SYSTEM VerticalCoalMill
  (* Version 1.0, Author, 4DIAC-Consortium *)
  APPLICATION Process
    FBS
      mF : REAL2REAL(IN := 1);
      F_MUL : F_MUL;
      F_ADD : F_ADD;
      F_ADD_0 : F_ADD;
      F_SUB : F_SUB;
      REAL2REAL_0 : REAL2REAL;
      REAL2REAL_0_0 : REAL2REAL;
      REAL2REAL_0_1 : REAL2REAL;
      a1 : REAL2REAL(IN := 0.5);
      m_SB : REAL2REAL(IN := 1);
      m_CB : REAL2REAL(IN := 1);
      E_CYCLE : E_CYCLE(DT := T#200ms);
      FB_INTEGRATE : FB_INTEGRATE(K := 1);
      REAL2REAL_0_1_0 : REAL2REAL;
      M_B2 : REAL2REAL;
      F_DIV : F_DIV;
      mBG : REAL2REAL;
      tauBG : REAL2REAL(IN := 0.5);
      MV_from_ESCADA : SUBSCRIBE_1(QI := 1, ID := 127.0.0.1:63100);
      PP_from_ESCADA1 : SUBSCRIBE_2(QI := 1, ID := 127.0.0.1:64100);
      START_Subscribe : SUBSCRIBE_1(QI := 1, ID := 127.0.0.1:10000);
      E_SWITCH_0 : E_SWITCH;
      m_BG : REAL2REAL(IN := 1);
      gamma1 : REAL2REAL(IN := 0.5);
      bJ : REAL2REAL(IN := 0.5);
      gammaJ : REAL2REAL(IN := 0.5);
      F_ADD_1 : F_ADD;
      REAL2REAL_2_0 : REAL2REAL;
      F_SUB_0 : F_SUB;
      FB_INTEGRATE_0 : FB_INTEGRATE(K := 1);
      REAL2REAL_2_0_0 : REAL2REAL;
      F_DIV_0 : F_DIV;
      tauGS : REAL2REAL(IN := 0.5);
      mGS : REAL2REAL;
      E_CYCLE_0 : E_CYCLE(DT := T#200ms);
      F_MUL_1 : F_MUL;
      F_MUL_1_2 : F_MUL;
      F_MUL_1_3 : F_MUL;
      REAL2REAL_2_0_3 : REAL2REAL;
      F_SUB_0_0 : F_SUB;
      REAL2REAL_2_0_3_0 : REAL2REAL;
      REAL2REAL_2_0_3_1 : REAL2REAL;
      REAL2REAL_2_0_3_0_0 : REAL2REAL;
      M_G2 : REAL2REAL;
      to_InputOutput1 : PUBLISH_2(QI := 1, ID := 127.0.0.1:62200);
      from_EclipseScada5 : SUBSCRIBE_4(QI := 1, ID := 127.0.0.1:64200);
      SUBSCRIBE_1_2 : SUBSCRIBE_1(QI := 1, ID := 127.0.0.1:20000);
      E_SWITCH_1 : E_SWITCH;
      m_air_inC : REAL2REAL(IN := 1);
      Cons1_0 : REAL2REAL(IN := 0.5959);
      F_MUL_2_1 : F_MUL;
      F_MUL_2_0_1 : F_MUL;
      REAL2REAL_2_1 : REAL2REAL;
      F_MUL_2_0_0_0 : F_MUL;
      Cons2_0 : REAL2REAL(IN := 22.69);
      REAL2REAL_2_2_1 : REAL2REAL;
      REAL2REAL_2_2_0_0 : REAL2REAL;
      F_SUB_1_0 : F_SUB;
      Cons3_0 : REAL2REAL(IN := 311.36);
      F_ADD_2_0 : F_ADD;
      REAL2REAL_2_2_0_1_0 : REAL2REAL;
      c2 : REAL2REAL;
      REAL2REAL_2_2_1_0_1 : REAL2REAL;
      F_SUB_2_1 : F_SUB;
      F_MUL_5_0 : F_MUL;
      cons4_0 : REAL2REAL(IN := 0.001);
      REAL2REAL_2_2_1_0_0_0 : REAL2REAL;
      d_min_0 : REAL2REAL(IN := 0.25);
      F_SUB_2_0_0 : F_SUB;
      d_max_0 : REAL2REAL(IN := 0.5);
      REAL2REAL_2_2_1_1_0 : REAL2REAL;
      REAL2REAL_2_2_1_2_0 : REAL2REAL;
      F_DIV_4 : F_DIV;
      m_SC : REAL2REAL(IN := 1);
      tau_CFU : REAL2REAL(IN := 0.5);
      tau_CB : REAL2REAL(IN := 0.5);
      m_AirIN : REAL2REAL(IN := 1);
      F_ADD_3_0 : F_ADD;
      REAL2REAL_21 : REAL2REAL;
      F_SUB_4_0 : F_SUB;
      REAL2REAL_8_0 : REAL2REAL;
      F_SUB_4_0_0 : F_SUB;
      REAL2REAL_8_0_0 : REAL2REAL;
      FB_INTEGRATE_2 : FB_INTEGRATE(K := 1);
      F_MUL_7 : F_MUL;
      REAL2REAL_10_0 : REAL2REAL;
      F_DIV_5 : F_DIV;
      mCFU : REAL2REAL;
      F_SUB_7_0 : F_SUB;
      REAL2REAL_10_0_0 : REAL2REAL(IN := 1);
      F_MUL_7_0 : F_MUL;
      REAL2REAL_10_1 : REAL2REAL;
      F_DIV_5_0 : F_DIV;
      mCB : REAL2REAL;
      REAL2REAL_10_0_0_0 : REAL2REAL;
      E_CYCLE_2 : E_CYCLE(DT := T#200ms);
      M_C2 : REAL2REAL;
      m_air_outC : REAL2REAL;
      to_InputOutput3 : PUBLISH_4(QI := 1, ID := 127.0.0.1:62400);
      SUBSCRIBE_1_3 : SUBSCRIBE_1(QI := 1, ID := 127.0.0.1:40000);
      E_SWITCH_2 : E_SWITCH;
      from_EclipseScada7 : SUBSCRIBE_4(QI := 1, ID := 127.0.0.1:64400);
      E_CYCLE_3 : E_CYCLE(DT := T#200ms);
      m_airS : REAL2REAL(IN := 1);
      Cp_a : REAL2REAL(IN := 0.5);
      T_m_air : REAL2REAL(IN := 25);
      F_MUL_0 : F_MUL;
      REAL2REAL_1_0 : REAL2REAL;
      F_MUL_8 : F_MUL;
      REAL2REAL_4_0 : REAL2REAL;
      m_CF : REAL2REAL(IN := 1);
      Satu : REAL2REAL(IN := 1);
      theta_FB : REAL2REAL(IN := 0.5);
      Cp : REAL2REAL(IN := 0.5);
      T_a : REAL2REAL(IN := 25);
      F_SUB_6 : F_SUB;
      F_MUL_9 : F_MUL;
      REAL2REAL_6_0 : REAL2REAL;
      F_MUL_10 : F_MUL;
      REAL2REAL_9_0 : REAL2REAL;
      REAL2REAL_11_0 : REAL2REAL;
      F_MUL_11 : F_MUL;
      REAL2REAL_12_0 : REAL2REAL;
      Cp_w : REAL2REAL(IN := 0.5);
      F_MUL_12 : F_MUL;
      F_MUL_13 : F_MUL;
      REAL2REAL_13_0 : REAL2REAL;
      REAL2REAL_14_0 : REAL2REAL;
      F_MUL_14 : F_MUL;
      REAL2REAL_15_0 : REAL2REAL;
      Hg : REAL2REAL(IN := 5);
      m_mois : REAL2REAL(IN := 1);
      h : REAL2REAL(IN := 0.5);
      v_t : REAL2REAL(IN := 0.5);
      F_MUL_13_0 : F_MUL;
      REAL2REAL_16_0 : REAL2REAL;
      F_MUL_17 : F_MUL;
      REAL2REAL_17_0 : REAL2REAL;
      K_loss : REAL2REAL(IN := 0.5);
      F_MUL_15_0 : F_MUL;
      REAL2REAL_18_0 : REAL2REAL;
      F_ADD_4 : F_ADD;
      REAL2REAL_19_0 : REAL2REAL;
      F_ADD_5 : F_ADD;
      REAL2REAL_20_0 : REAL2REAL;
      F_SUB_8 : F_SUB;
      REAL2REAL_21_0 : REAL2REAL;
      F_ADD_6 : F_ADD;
      REAL2REAL_22_0 : REAL2REAL;
      F_ADD_7 : F_ADD;
      REAL2REAL_23_0 : REAL2REAL;
      m_CFU : REAL2REAL(IN := 1);
      Satu1 : REAL2REAL(IN := 1);
      theta_out : REAL2REAL(IN := 0.5);
      Cp_c : REAL2REAL(IN := 0.5);
      F_SUB_9 : F_SUB;
      REAL2REAL_24_0 : REAL2REAL;
      F_MUL_16_0 : F_MUL;
      REAL2REAL_25_0 : REAL2REAL;
      F_MUL_18_0 : F_MUL;
      REAL2REAL_26_0 : REAL2REAL;
      F_MUL_19_0 : F_MUL;
      REAL2REAL_27_0 : REAL2REAL;
      Cp_w1 : REAL2REAL(IN := 0.5);
      F_MUL_20_0 : F_MUL;
      REAL2REAL_29_0 : REAL2REAL;
      F_MUL_21_0 : F_MUL;
      REAL2REAL_30_0 : REAL2REAL;
      F_MUL_22_0 : F_MUL;
      REAL2REAL_31_0 : REAL2REAL;
      Cp1 : REAL2REAL(IN := 0.5);
      F_MUL_24_0 : F_MUL;
      REAL2REAL_28_0 : REAL2REAL;
      F_MUL_25_0 : F_MUL;
      REAL2REAL_32_0 : REAL2REAL;
      K_loss1 : REAL2REAL(IN := 1);
      F_MUL_23_0 : F_MUL;
      REAL2REAL_33_0 : REAL2REAL;
      REAL2REAL_34_0 : REAL2REAL;
      F_ADD_8 : F_ADD;
      REAL2REAL_35_0 : REAL2REAL;
      F_ADD_9 : F_ADD;
      REAL2REAL_36_0 : REAL2REAL;
      F_SUB_11 : F_SUB;
      REAL2REAL_37_0 : REAL2REAL;
      M_met : REAL2REAL(IN := 1);
      Cp_met : REAL2REAL(IN := 0.5);
      F_MUL_26_0 : F_MUL;
      REAL2REAL_38_0 : REAL2REAL;
      M_B : REAL2REAL(IN := 1);
      M_G : REAL2REAL(IN := 1);
      M_C : REAL2REAL(IN := 1);
      F_ADD_10 : F_ADD;
      REAL2REAL_39_0 : REAL2REAL;
      F_ADD_11 : F_ADD;
      REAL2REAL_40_0 : REAL2REAL;
      REAL2REAL_41_0 : REAL2REAL;
      Satu2 : REAL2REAL(IN := 1);
      theta_acc : REAL2REAL(IN := 0.5);
      F_SUB_12 : F_SUB;
      Cp_c1 : REAL2REAL(IN := 0.5);
      F_MUL_27_0 : F_MUL;
      REAL2REAL_42_0 : REAL2REAL;
      F_MUL_28_0 : F_MUL;
      REAL2REAL_43_0 : REAL2REAL;
      F_ADD_12 : F_ADD;
      REAL2REAL_44_0 : REAL2REAL;
      F_ADD_13 : F_ADD;
      REAL2REAL_45_0 : REAL2REAL;
      F_MUL_29_0 : F_MUL;
      REAL2REAL_46_0 : REAL2REAL;
      Cp_w2 : REAL2REAL(IN := 0.5);
      F_MUL_30_0 : F_MUL;
      REAL2REAL_47_0 : REAL2REAL;
      F_ADD_14 : F_ADD;
      REAL2REAL_48_0 : REAL2REAL;
      F_ADD_15 : F_ADD;
      REAL2REAL_49_0 : REAL2REAL;
      F_DIV_6 : F_DIV;
      dT_out : REAL2REAL;
      FB_INTEGRATE_3 : FB_INTEGRATE(K := 1);
      T_out : REAL2REAL;
      to_InputOutput4 : PUBLISH_1(QI := 1, ID := 127.0.0.1:62500);
      from_EclipseScada2 : SUBSCRIBE_4(QI := 1, ID := 127.0.0.1:63500);
      SUBSCRIBE_1_4 : SUBSCRIBE_1(QI := 1, ID := 127.0.0.1:50000);
      E_SWITCH_3 : E_SWITCH;
      from_EclipseScada8 : SUBSCRIBE_6(QI := 1, ID := 127.0.0.1:64501);
      from_EclipseScada9 : SUBSCRIBE_6(QI := 1, ID := 127.0.0.1:64502);
      from_EclipseScada10 : SUBSCRIBE_4(QI := 1, ID := 127.0.0.1:64503);
      F_ADD_3 : F_ADD;
      E_CYCLE_4 : E_CYCLE(DT := T#200ms);
      K_auf : REAL2REAL(IN := 0.5);
      m_airS1 : REAL2REAL(IN := 1);
      F_MUL_31 : F_MUL;
      REAL2REAL_52 : REAL2REAL;
      F_MUL_32 : F_MUL;
      REAL2REAL_53 : REAL2REAL;
      K_c : REAL2REAL(IN := 0.5);
      M_B1 : REAL2REAL(IN := 1);
      M_G1 : REAL2REAL(IN := 1);
      F_ADD_16 : F_ADD;
      REAL2REAL_54 : REAL2REAL;
      m_airS2 : REAL2REAL(IN := 1);
      F_MUL_33 : F_MUL;
      REAL2REAL_55 : REAL2REAL;
      F_MUL_34 : F_MUL;
      REAL2REAL_56 : REAL2REAL;
      F_MUL_35 : F_MUL;
      REAL2REAL_57 : REAL2REAL;
      K_ce : REAL2REAL(IN := 0.5);
      M_S : REAL2REAL(IN := 1);
      M_C1 : REAL2REAL(IN := 1);
      m_airS3 : REAL2REAL(IN := 1);
      F_MUL_36 : F_MUL;
      REAL2REAL_58 : REAL2REAL;
      F_ADD_17 : F_ADD;
      REAL2REAL_59 : REAL2REAL;
      F_MUL_37 : F_MUL;
      REAL2REAL_60 : REAL2REAL;
      F_MUL_38 : F_MUL;
      REAL2REAL_61 : REAL2REAL;
      F_ADD_18 : F_ADD;
      REAL2REAL_62 : REAL2REAL;
      F_ADD_19 : F_ADD;
      dP_mill : REAL2REAL;
      to_InputOutput5 : PUBLISH_1(QI := 1, ID := 127.0.0.1:62600);
      SUBSCRIBE_1_5 : SUBSCRIBE_1(QI := 1, ID := 127.0.0.1:60000);
      E_SWITCH_4 : E_SWITCH;
      from_EclipseScada11 : SUBSCRIBE_3(QI := 1, ID := 127.0.0.1:64600);
      K_power : REAL2REAL(IN := 0.5);
      M_G3 : REAL2REAL(IN := 2);
      w : REAL2REAL(IN := 1);
      N_rol : REAL2REAL(IN := 0.5);
      F_MUL_39 : F_MUL;
      REAL2REAL_50 : REAL2REAL;
      F_MUL_40 : F_MUL;
      REAL2REAL_51 : REAL2REAL;
      F_MUL_41 : F_MUL;
      REAL2REAL_63 : REAL2REAL;
      P_load : REAL2REAL(IN := 2);
      F_ADD_20 : F_ADD;
      REAL2REAL_64 : REAL2REAL;
      M_on : REAL2REAL(IN := 1);
      F_MUL_42 : F_MUL;
      P_total : REAL2REAL;
      M_v : REAL2REAL(IN := 0.5);
      P_f : REAL2REAL(IN := 0.5);
      F_MUL_43 : F_MUL;
      REAL2REAL_66 : REAL2REAL;
      F_DIV_7 : F_DIV;
      I_total : REAL2REAL;
      K_g : REAL2REAL(IN := 0.5);
      F_MUL_44 : F_MUL;
      Hg1 : REAL2REAL;
      E_CYCLE_5 : E_CYCLE(DT := T#200ms);
      to_InputOutput6 : PUBLISH_3(QI := 1, ID := 127.0.0.1:62700);
      from_EclipseScada3 : SUBSCRIBE_1(QI := 1, ID := 127.0.0.1:63700);
      SUBSCRIBE_1_6 : SUBSCRIBE_1(QI := 1, ID := 127.0.0.1:70000);
      E_SWITCH_5 : E_SWITCH;
      from_EclipseScada12 : SUBSCRIBE_4(QI := 1, ID := 127.0.0.1:64701);
      from_EclipseScada13 : SUBSCRIBE_3(QI := 1, ID := 127.0.0.1:64702);
      m_air_inS_plus_noise : REAL2REAL;
      Cons1 : REAL2REAL(IN := 0.5728);
      F_MUL_2 : F_MUL;
      F_MUL_2_0 : F_MUL;
      REAL2REAL_2 : REAL2REAL;
      F_MUL_2_0_0 : F_MUL;
      Cons2 : REAL2REAL(IN := 14.307);
      REAL2REAL_2_2 : REAL2REAL;
      REAL2REAL_2_2_0 : REAL2REAL;
      F_SUB_1 : F_SUB;
      Cons3 : REAL2REAL(IN := 180.22);
      F_ADD_2 : F_ADD;
      REAL2REAL_2_2_0_1 : REAL2REAL;
      c1 : REAL2REAL;
      REAL2REAL_2_2_1_0 : REAL2REAL;
      F_SUB_2 : F_SUB;
      F_MUL_5 : F_MUL;
      cons4 : REAL2REAL(IN := 0.001);
      REAL2REAL_2_2_1_0_0 : REAL2REAL;
      d_min : REAL2REAL(IN := 0.25);
      F_SUB_2_0 : F_SUB;
      d_max : REAL2REAL(IN := 0.5);
      REAL2REAL_2_2_1_1 : REAL2REAL;
      REAL2REAL_2_2_1_2 : REAL2REAL;
      m_GS : REAL2REAL(IN := 1);
      rho : REAL2REAL(IN := 0.5);
      nu_acc : REAL2REAL(IN := 0.5);
      F_MUL_3_0 : F_MUL;
      F_MUL_4_0 : F_MUL;
      REAL2REAL_5_0 : REAL2REAL;
      m_mois1 : REAL2REAL;
      F_SUB_3_0 : F_SUB;
      REAL2REAL_5_0_0 : REAL2REAL;
      F_SUB_3_0_0 : F_SUB;
      REAL2REAL_5_0_0_0 : REAL2REAL;
      F_SUB_3_0_0_0 : F_SUB;
      REAL2REAL_5_0_0_0_0 : REAL2REAL;
      FB_INTEGRATE_1 : FB_INTEGRATE(K := 1);
      F_MUL_6_0 : F_MUL;
      REAL2REAL_7_0 : REAL2REAL;
      tauSC : REAL2REAL(IN := 0.5);
      tauSB : REAL2REAL(IN := 0.5);
      REAL2REAL_3_0 : REAL2REAL(IN := 1);
      F_SUB_5_0 : F_SUB;
      F_MUL_6_0_0 : F_MUL;
      REAL2REAL_7_0_0 : REAL2REAL;
      REAL2REAL_7_1 : REAL2REAL;
      F_DIV_1 : F_DIV;
      F_DIV_2 : F_DIV;
      mSC : REAL2REAL;
      mSB : REAL2REAL;
      E_CYCLE_1 : E_CYCLE(DT := T#200ms);
      F_DIV_3 : F_DIV;
      M_S1 : REAL2REAL;
      m_air_outS : REAL2REAL;
      m_air_inS : REAL2REAL(IN := 1);
      to_InputOutput2 : PUBLISH_5(QI := 1, ID := 127.0.0.1:62300);
      from_EclipseScada1 : SUBSCRIBE_1(QI := 1, ID := 127.0.0.1:63300);
      from_EclipseScada6 : SUBSCRIBE_6(QI := 1, ID := 127.0.0.1:64300);
      SUBSCRIBE_1_0 : SUBSCRIBE_1(QI := 1, ID := 127.0.0.1:30000);
      E_SWITCH : E_SWITCH;
    END_FBS
    EVENT_CONNECTIONS
       TO ;
       TO ;
       TO ;
       TO ;
      M_B2.CNF TO F_DIV.REQ;
      FB_INTEGRATE.CNF TO M_B2.REQ;
      F_SUB.CNF TO REAL2REAL_0_1_0.REQ;
      F_MUL.CNF TO REAL2REAL_0.REQ;
      REAL2REAL_0_1_0.CNF TO FB_INTEGRATE.REQ;
      F_ADD_0.CNF TO REAL2REAL_0_1.REQ;
      F_ADD.CNF TO REAL2REAL_0_0.REQ;
      REAL2REAL_0.CNF TO F_ADD.REQ;
      E_CYCLE.EO TO m_SB.REQ;
      REAL2REAL_0_0.CNF TO F_ADD_0.REQ;
      REAL2REAL_0_1.CNF TO F_SUB.REQ;
      E_CYCLE.EO TO tauBG.REQ;
      E_CYCLE.EO TO mF.REQ;
      E_CYCLE.EO TO m_CB.REQ;
      F_DIV.CNF TO mBG.REQ;
      E_CYCLE.EO TO a1.REQ;
      mF.CNF TO F_MUL.REQ;
      START.COLD TO FB_INTEGRATE.INIT;
      START.WARM TO FB_INTEGRATE.INIT;
      START.COLD TO MV_from_ESCADA.INIT;
      START.WARM TO MV_from_ESCADA.INIT;
      START.COLD TO PP_from_ESCADA1.INIT;
      START.WARM TO PP_from_ESCADA1.INIT;
      START_Subscribe.IND TO E_SWITCH_0.EI;
      E_SWITCH_0.EO1 TO E_CYCLE.START;
      START.COLD TO START_Subscribe.INIT;
      START.WARM TO START_Subscribe.INIT;
      REAL2REAL_2_0.CNF TO F_SUB_0.REQ;
      m_BG.CNF TO F_ADD_1.REQ;
      E_CYCLE_0.EO TO tauGS.REQ;
      F_MUL_1_3.CNF TO REAL2REAL_2_0_3_1.REQ;
      F_SUB_0_0.CNF TO REAL2REAL_2_0_3_0_0.REQ;
      E_CYCLE_0.EO TO bJ.REQ;
      F_ADD_1.CNF TO REAL2REAL_2_0.REQ;
      REAL2REAL_2_0_3.CNF TO F_MUL_1_3.REQ;
      REAL2REAL_2_0_0.CNF TO FB_INTEGRATE_0.REQ;
      F_DIV_0.CNF TO mGS.REQ;
      REAL2REAL_2_0_3_0.CNF TO F_SUB_0_0.REQ;
      F_MUL_1_2.CNF TO REAL2REAL_2_0_3.REQ;
      FB_INTEGRATE_0.CNF TO F_MUL_1_2.REQ;
      FB_INTEGRATE_0.CNF TO F_DIV_0.REQ;
      E_CYCLE_0.EO TO m_BG.REQ;
      FB_INTEGRATE_0.CNF TO M_G2.REQ;
      FB_INTEGRATE_0.CNF TO F_MUL_1.REQ;
      F_MUL_1.CNF TO REAL2REAL_2_0_3_0.REQ;
      F_SUB_0.CNF TO REAL2REAL_2_0_0.REQ;
      E_CYCLE_0.EO TO gammaJ.REQ;
      E_CYCLE_0.EO TO gamma1.REQ;
      START.COLD TO FB_INTEGRATE_0.INIT;
      START.WARM TO FB_INTEGRATE_0.INIT;
      mGS.CNF TO to_InputOutput1.REQ;
      FB_INTEGRATE_0.INITO TO to_InputOutput1.INIT;
      START.COLD TO from_EclipseScada5.INIT;
      START.WARM TO from_EclipseScada5.INIT;
      SUBSCRIBE_1_2.IND TO E_SWITCH_1.EI;
      E_SWITCH_1.EO1 TO E_CYCLE_0.START;
      START.COLD TO SUBSCRIBE_1_2.INIT;
      START.WARM TO SUBSCRIBE_1_2.INIT;
      REAL2REAL_2_2_0_1_0.CNF TO F_ADD_2_0.REQ;
      FB_INTEGRATE_2.CNF TO M_C2.REQ;
      E_CYCLE_2.EO TO m_SC.REQ;
      REAL2REAL_10_0.CNF TO F_DIV_5.REQ;
      E_CYCLE_2.EO TO tau_CFU.REQ;
      F_MUL_2_0_1.CNF TO REAL2REAL_2_1.REQ;
      REAL2REAL_21.CNF TO F_SUB_4_0.REQ;
      REAL2REAL_10_0_0_0.CNF TO F_MUL_7_0.REQ;
      REAL2REAL_2_2_1_0_0_0.CNF TO F_SUB_2_1.REQ;
      REAL2REAL_8_0_0.CNF TO FB_INTEGRATE_2.REQ;
      Cons2_0.CNF TO F_MUL_2_0_0_0.REQ;
      F_SUB_2_0_0.CNF TO REAL2REAL_2_2_1_1_0.REQ;
      F_SUB_2_1.CNF TO REAL2REAL_2_2_1_2_0.REQ;
      F_DIV_5_0.CNF TO mCB.REQ;
      E_CYCLE_2.EO TO Cons1_0.REQ;
      F_ADD_2_0.CNF TO cons4_0.REQ;
      FB_INTEGRATE_2.CNF TO REAL2REAL_10_0_0_0.REQ;
      m_air_inC.CNF TO m_air_outC.REQ;
      F_MUL_2_1.CNF TO REAL2REAL_2_2_0_0.REQ;
      c2.CNF TO REAL2REAL_10_0_0.REQ;
      F_DIV_5.CNF TO mCFU.REQ;
      F_SUB_1_0.CNF TO REAL2REAL_2_2_0_1_0.REQ;
      F_SUB_4_0.CNF TO REAL2REAL_8_0.REQ;
      E_CYCLE_2.EO TO m_air_inC.REQ;
      c2.CNF TO F_SUB_7_0.REQ;
      F_MUL_5_0.CNF TO d_min_0.REQ;
      REAL2REAL_8_0.CNF TO F_SUB_4_0_0.REQ;
      FB_INTEGRATE_2.CNF TO F_MUL_7.REQ;
      E_CYCLE_2.EO TO Cons2_0.REQ;
      F_DIV_4.CNF TO c2.REQ;
      m_air_inC.CNF TO F_MUL_2_0_1.REQ;
      F_ADD_3_0.CNF TO REAL2REAL_21.REQ;
      F_MUL_7_0.CNF TO REAL2REAL_10_1.REQ;
      F_MUL_2_0_0_0.CNF TO REAL2REAL_2_2_1.REQ;
      REAL2REAL_2_2_1_0_0_0.CNF TO F_SUB_2_0_0.REQ;
      F_SUB_4_0_0.CNF TO REAL2REAL_8_0_0.REQ;
      REAL2REAL_2_1.CNF TO F_MUL_2_1.REQ;
      E_CYCLE_2.EO TO m_AirIN.REQ;
      F_MUL_7.CNF TO REAL2REAL_10_0.REQ;
      REAL2REAL_2_2_1_0_1.CNF TO F_MUL_5_0.REQ;
      m_AirIN.CNF TO F_ADD_3_0.REQ;
      REAL2REAL_2_2_1_2_0.CNF TO F_DIV_4.REQ;
      REAL2REAL_10_1.CNF TO F_DIV_5_0.REQ;
      F_ADD_2_0.CNF TO REAL2REAL_2_2_1_0_1.REQ;
      E_CYCLE_2.EO TO Cons3_0.REQ;
      F_MUL_5_0.CNF TO d_max_0.REQ;
      E_CYCLE_2.EO TO tau_CB.REQ;
      REAL2REAL_2_2_0_0.CNF TO F_SUB_1_0.REQ;
      F_MUL_5_0.CNF TO REAL2REAL_2_2_1_0_0_0.REQ;
      START.COLD TO FB_INTEGRATE_2.INIT;
      START.WARM TO FB_INTEGRATE_2.INIT;
      mCFU.CNF TO to_InputOutput3.REQ;
      FB_INTEGRATE_2.INITO TO to_InputOutput3.INIT;
      SUBSCRIBE_1_3.IND TO E_SWITCH_2.EI;
      E_SWITCH_2.EO1 TO E_CYCLE_2.START;
      START.COLD TO SUBSCRIBE_1_3.INIT;
      START.WARM TO SUBSCRIBE_1_3.INIT;
      START.COLD TO from_EclipseScada7.INIT;
      START.WARM TO from_EclipseScada7.INIT;
      F_MUL_21_0.CNF TO REAL2REAL_30_0.REQ;
      dT_out.CNF TO FB_INTEGRATE_3.REQ;
      F_MUL_30_0.CNF TO REAL2REAL_47_0.REQ;
      Cp_w.CNF TO F_MUL_13.REQ;
      F_MUL_11.CNF TO REAL2REAL_12_0.REQ;
      F_MUL_28_0.CNF TO REAL2REAL_43_0.REQ;
      F_SUB_6.CNF TO REAL2REAL_6_0.REQ;
      F_MUL_20_0.CNF TO REAL2REAL_29_0.REQ;
      F_ADD_13.CNF TO REAL2REAL_45_0.REQ;
      E_CYCLE_3.EO TO M_B.REQ;
      Cp_c.CNF TO F_MUL_18_0.REQ;
      REAL2REAL_37_0.CNF TO F_DIV_6.REQ;
      K_loss.CNF TO F_MUL_15_0.REQ;
      REAL2REAL_42_0.CNF TO F_MUL_28_0.REQ;
      F_MUL_16_0.CNF TO REAL2REAL_25_0.REQ;
      REAL2REAL_40_0.CNF TO F_MUL_27_0.REQ;
      Satu.CNF TO F_SUB_6.REQ;
      E_CYCLE_3.EO TO Cp_c.REQ;
      M_met.CNF TO F_MUL_26_0.REQ;
      F_ADD_15.CNF TO REAL2REAL_49_0.REQ;
      M_B.CNF TO F_ADD_10.REQ;
      F_MUL_12.CNF TO REAL2REAL_13_0.REQ;
      F_MUL_17.CNF TO REAL2REAL_17_0.REQ;
      E_CYCLE_3.EO TO theta_acc.REQ;
      F_MUL_22_0.CNF TO REAL2REAL_31_0.REQ;
      E_CYCLE_3.EO TO h.REQ;
      E_CYCLE_3.EO TO M_C.REQ;
      F_ADD_4.CNF TO REAL2REAL_19_0.REQ;
      E_CYCLE_3.EO TO Satu.REQ;
      REAL2REAL_22_0.CNF TO F_ADD_7.REQ;
      E_CYCLE_3.EO TO T_a.REQ;
      m_mois.CNF TO F_MUL_13_0.REQ;
      m_airS.CNF TO F_MUL_0.REQ;
      E_CYCLE_3.EO TO M_met.REQ;
      m_CF.CNF TO F_MUL_12.REQ;
      F_MUL_29_0.CNF TO REAL2REAL_46_0.REQ;
      F_MUL_18_0.CNF TO REAL2REAL_26_0.REQ;
      F_ADD_12.CNF TO REAL2REAL_44_0.REQ;
      F_SUB_9.CNF TO REAL2REAL_24_0.REQ;
      E_CYCLE_3.EO TO Cp1.REQ;
      F_MUL_23_0.CNF TO REAL2REAL_33_0.REQ;
      REAL2REAL_44_0.CNF TO F_ADD_13.REQ;
      REAL2REAL_29_0.CNF TO F_MUL_22_0.REQ;
      REAL2REAL_25_0.CNF TO F_MUL_19_0.REQ;
      E_CYCLE_3.EO TO Cp.REQ;
      E_CYCLE_3.EO TO m_CFU.REQ;
      E_CYCLE_3.EO TO Cp_met.REQ;
      REAL2REAL_16_0.CNF TO F_MUL_17.REQ;
      REAL2REAL_46_0.CNF TO F_MUL_30_0.REQ;
      REAL2REAL_48_0.CNF TO F_ADD_15.REQ;
      E_CYCLE_3.EO TO m_CF.REQ;
      F_MUL_14.CNF TO REAL2REAL_15_0.REQ;
      F_MUL_9.CNF TO REAL2REAL_9_0.REQ;
      F_MUL_8.CNF TO REAL2REAL_4_0.REQ;
      E_CYCLE_3.EO TO m_mois.REQ;
      E_CYCLE_3.EO TO theta_out.REQ;
      REAL2REAL_17_0.CNF TO F_SUB_8.REQ;
      F_ADD_7.CNF TO REAL2REAL_23_0.REQ;
      Cp1.CNF TO F_MUL_24_0.REQ;
      F_SUB_8.CNF TO REAL2REAL_21_0.REQ;
      REAL2REAL_1_0.CNF TO F_MUL_8.REQ;
      E_CYCLE_3.EO TO Cp_c1.REQ;
      E_CYCLE_3.EO TO T_m_air.REQ;
      F_MUL_19_0.CNF TO REAL2REAL_27_0.REQ;
      REAL2REAL_15_0.CNF TO F_ADD_5.REQ;
      E_CYCLE_3.EO TO m_airS.REQ;
      F_MUL_24_0.CNF TO REAL2REAL_28_0.REQ;
      REAL2REAL_28_0.CNF TO F_MUL_25_0.REQ;
      F_MUL_13.CNF TO REAL2REAL_14_0.REQ;
      Satu2.CNF TO F_SUB_12.REQ;
      F_MUL_15_0.CNF TO REAL2REAL_18_0.REQ;
      REAL2REAL_9_0.CNF TO F_MUL_11.REQ;
      E_CYCLE_3.EO TO theta_FB.REQ;
      E_CYCLE_3.EO TO Cp_a.REQ;
      M_B.CNF TO F_ADD_12.REQ;
      E_CYCLE_3.EO TO M_G.REQ;
      E_CYCLE_3.EO TO Satu2.REQ;
      REAL2REAL_34_0.CNF TO F_ADD_9.REQ;
      E_CYCLE_3.EO TO K_loss.REQ;
      REAL2REAL_13_0.CNF TO F_MUL_14.REQ;
      REAL2REAL_6_0.CNF TO F_MUL_9.REQ;
      REAL2REAL_24_0.CNF TO F_MUL_16_0.REQ;
      F_MUL_0.CNF TO REAL2REAL_1_0.REQ;
      F_ADD_8.CNF TO REAL2REAL_35_0.REQ;
      E_CYCLE_3.EO TO Cp_w1.REQ;
      REAL2REAL_20_0.CNF TO F_ADD_6.REQ;
      E_CYCLE_3.EO TO K_loss1.REQ;
      F_MUL_25_0.CNF TO REAL2REAL_32_0.REQ;
      m_CFU.CNF TO F_MUL_20_0.REQ;
      REAL2REAL_39_0.CNF TO F_ADD_11.REQ;
      F_MUL_13_0.CNF TO REAL2REAL_16_0.REQ;
      F_ADD_11.CNF TO REAL2REAL_40_0.REQ;
      F_DIV_6.CNF TO dT_out.REQ;
      REAL2REAL_32_0.CNF TO F_ADD_8.REQ;
      FB_INTEGRATE_3.CNF TO T_out.REQ;
      K_loss1.CNF TO F_MUL_23_0.REQ;
      F_MUL_10.CNF TO REAL2REAL_11_0.REQ;
      F_MUL_27_0.CNF TO REAL2REAL_42_0.REQ;
      F_ADD_10.CNF TO REAL2REAL_39_0.REQ;
      F_ADD_14.CNF TO REAL2REAL_48_0.REQ;
      Cp_w1.CNF TO F_MUL_21_0.REQ;
      F_ADD_6.CNF TO REAL2REAL_22_0.REQ;
      F_SUB_11.CNF TO REAL2REAL_37_0.REQ;
      F_ADD_9.CNF TO REAL2REAL_36_0.REQ;
      E_CYCLE_3.EO TO Cp_w.REQ;
      REAL2REAL_4_0.CNF TO F_ADD_4.REQ;
      Cp.CNF TO F_MUL_10.REQ;
      Satu1.CNF TO F_SUB_9.REQ;
      REAL2REAL_45_0.CNF TO F_MUL_29_0.REQ;
      F_SUB_12.CNF TO REAL2REAL_41_0.REQ;
      REAL2REAL_43_0.CNF TO F_ADD_14.REQ;
      E_CYCLE_3.EO TO Satu1.REQ;
      REAL2REAL_23_0.CNF TO F_SUB_11.REQ;
      E_CYCLE_3.EO TO Cp_w2.REQ;
      F_ADD_5.CNF TO REAL2REAL_20_0.REQ;
      F_MUL_26_0.CNF TO REAL2REAL_38_0.REQ;
      E_CYCLE_3.EO TO v_t.REQ;
      START.COLD TO FB_INTEGRATE_3.INIT;
      START.WARM TO FB_INTEGRATE_3.INIT;
      E_CYCLE_3.EO TO Hg.REQ;
      T_out.CNF TO to_InputOutput4.REQ;
      FB_INTEGRATE_3.INITO TO to_InputOutput4.INIT;
      START.COLD TO from_EclipseScada2.INIT;
      START.WARM TO from_EclipseScada2.INIT;
      SUBSCRIBE_1_4.IND TO E_SWITCH_3.EI;
      E_SWITCH_3.EO1 TO E_CYCLE_3.START;
      START.COLD TO SUBSCRIBE_1_4.INIT;
      START.WARM TO SUBSCRIBE_1_4.INIT;
      START.COLD TO from_EclipseScada8.INIT;
      START.WARM TO from_EclipseScada8.INIT;
      START.COLD TO from_EclipseScada9.INIT;
      START.WARM TO from_EclipseScada9.INIT;
      START.COLD TO from_EclipseScada10.INIT;
      START.WARM TO from_EclipseScada10.INIT;
      REAL2REAL_27_0.CNF TO F_ADD_3.REQ;
      F_ADD_3.CNF TO REAL2REAL_34_0.REQ;
      REAL2REAL_62.CNF TO F_ADD_19.REQ;
      E_CYCLE_4.EO TO m_airS2.REQ;
      F_ADD_17.CNF TO REAL2REAL_59.REQ;
      F_MUL_36.CNF TO REAL2REAL_58.REQ;
      REAL2REAL_52.CNF TO F_MUL_32.REQ;
      REAL2REAL_54.CNF TO F_MUL_34.REQ;
      F_MUL_35.CNF TO REAL2REAL_57.REQ;
      E_CYCLE_4.EO TO K_ce.REQ;
      E_CYCLE_4.EO TO M_C1.REQ;
      E_CYCLE_4.EO TO m_airS1.REQ;
      REAL2REAL_56.CNF TO F_MUL_35.REQ;
      M_S.CNF TO F_ADD_17.REQ;
      E_CYCLE_4.EO TO M_G1.REQ;
      E_CYCLE_4.EO TO M_S.REQ;
      F_ADD_19.CNF TO dP_mill.REQ;
      F_MUL_34.CNF TO REAL2REAL_56.REQ;
      F_MUL_38.CNF TO REAL2REAL_61.REQ;
      F_MUL_32.CNF TO REAL2REAL_53.REQ;
      REAL2REAL_60.CNF TO F_MUL_38.REQ;
      m_airS1.CNF TO F_MUL_31.REQ;
      F_ADD_16.CNF TO REAL2REAL_54.REQ;
      m_airS2.CNF TO F_MUL_33.REQ;
      M_B1.CNF TO F_ADD_16.REQ;
      E_CYCLE_4.EO TO K_auf.REQ;
      F_ADD_18.CNF TO REAL2REAL_62.REQ;
      F_MUL_37.CNF TO REAL2REAL_60.REQ;
      E_CYCLE_4.EO TO m_airS3.REQ;
      F_MUL_31.CNF TO REAL2REAL_52.REQ;
      REAL2REAL_57.CNF TO F_ADD_18.REQ;
      E_CYCLE_4.EO TO M_B1.REQ;
      F_MUL_33.CNF TO REAL2REAL_55.REQ;
      E_CYCLE_4.EO TO K_c.REQ;
      m_airS3.CNF TO F_MUL_36.REQ;
      REAL2REAL_59.CNF TO F_MUL_37.REQ;
      dP_mill.CNF TO to_InputOutput5.REQ;
      START.COLD TO to_InputOutput5.INIT;
      START.WARM TO to_InputOutput5.INIT;
      SUBSCRIBE_1_5.IND TO E_SWITCH_4.EI;
      E_SWITCH_4.EO1 TO E_CYCLE_4.START;
      START.COLD TO SUBSCRIBE_1_5.INIT;
      START.WARM TO SUBSCRIBE_1_5.INIT;
      START.COLD TO from_EclipseScada11.INIT;
      START.WARM TO from_EclipseScada11.INIT;
      E_CYCLE_5.EO TO M_G3.REQ;
      E_CYCLE_5.EO TO N_rol.REQ;
      w.CNF TO F_MUL_40.REQ;
      E_CYCLE_5.EO TO K_power.REQ;
      M_v.CNF TO F_MUL_43.REQ;
      P_total.CNF TO F_DIV_7.REQ;
      F_DIV_7.CNF TO I_total.REQ;
      E_CYCLE_5.EO TO P_load.REQ;
      E_CYCLE_5.EO TO M_on.REQ;
      M_G3.CNF TO F_MUL_39.REQ;
      E_CYCLE_5.EO TO K_g.REQ;
      REAL2REAL_50.CNF TO F_MUL_41.REQ;
      F_MUL_40.CNF TO REAL2REAL_51.REQ;
      E_CYCLE_5.EO TO w.REQ;
      I_total.CNF TO F_MUL_44.REQ;
      F_MUL_43.CNF TO REAL2REAL_66.REQ;
      E_CYCLE_5.EO TO M_v.REQ;
      F_MUL_42.CNF TO P_total.REQ;
      F_MUL_41.CNF TO REAL2REAL_63.REQ;
      F_MUL_39.CNF TO REAL2REAL_50.REQ;
      F_MUL_44.CNF TO Hg1.REQ;
      REAL2REAL_63.CNF TO F_ADD_20.REQ;
      REAL2REAL_64.CNF TO F_MUL_42.REQ;
      E_CYCLE_5.EO TO P_f.REQ;
      F_ADD_20.CNF TO REAL2REAL_64.REQ;
      Hg1.CNF TO to_InputOutput6.REQ;
      START.COLD TO to_InputOutput6.INIT;
      START.WARM TO to_InputOutput6.INIT;
      START.COLD TO from_EclipseScada3.INIT;
      START.WARM TO from_EclipseScada3.INIT;
      SUBSCRIBE_1_6.IND TO E_SWITCH_5.EI;
      E_SWITCH_5.EO1 TO E_CYCLE_5.START;
      START.COLD TO SUBSCRIBE_1_6.INIT;
      START.WARM TO SUBSCRIBE_1_6.INIT;
      START.COLD TO from_EclipseScada12.INIT;
      START.WARM TO from_EclipseScada12.INIT;
      START.COLD TO from_EclipseScada13.INIT;
      START.WARM TO from_EclipseScada13.INIT;
      REAL2REAL_2_2_1_0_0.CNF TO F_SUB_2.REQ;
      REAL2REAL_5_0_0_0.CNF TO F_SUB_3_0_0_0.REQ;
      E_CYCLE_1.EO TO tauSC.REQ;
      REAL2REAL_5_0_0_0_0.CNF TO REAL2REAL_3_0.REQ;
      F_SUB_2.CNF TO REAL2REAL_2_2_1_2.REQ;
      F_MUL_5.CNF TO d_min.REQ;
      E_CYCLE_1.EO TO m_GS.REQ;
      rho.CNF TO F_MUL_3_0.REQ;
      REAL2REAL_7_1.CNF TO F_DIV_2.REQ;
      REAL2REAL_2_2_0_1.CNF TO F_ADD_2.REQ;
      E_CYCLE_1.EO TO Cons2.REQ;
      F_MUL_5.CNF TO d_max.REQ;
      Cons2.CNF TO F_MUL_2_0_0.REQ;
      E_CYCLE_1.EO TO rho.REQ;
      F_MUL_5.CNF TO REAL2REAL_2_2_1_0_0.REQ;
      F_SUB_1.CNF TO REAL2REAL_2_2_0_1.REQ;
      E_CYCLE_1.EO TO nu_acc.REQ;
      m_air_inS_plus_noise.CNF TO F_MUL_2_0.REQ;
      m_GS.CNF TO F_MUL_4_0.REQ;
      F_DIV_2.CNF TO mSB.REQ;
      REAL2REAL_2_2_0.CNF TO F_SUB_1.REQ;
      m_mois1.CNF TO F_SUB_3_0.REQ;
      F_SUB_2_0.CNF TO REAL2REAL_2_2_1_1.REQ;
      F_MUL_6_0.CNF TO REAL2REAL_7_0.REQ;
      F_SUB_3_0_0_0.CNF TO REAL2REAL_5_0_0_0_0.REQ;
      F_MUL_4_0.CNF TO m_mois1.REQ;
      E_CYCLE_1.EO TO Cons1.REQ;
      E_CYCLE_1.EO TO m_air_inS.REQ;
      F_MUL_2_0_0.CNF TO REAL2REAL_2_2.REQ;
      m_air_inS_plus_noise.CNF TO m_air_outS.REQ;
      E_CYCLE_1.EO TO tauSB.REQ;
      REAL2REAL_2_2_1_0.CNF TO F_MUL_5.REQ;
      FB_INTEGRATE_1.CNF TO M_S1.REQ;
      F_DIV_3.CNF TO c1.REQ;
      F_MUL_6_0_0.CNF TO REAL2REAL_7_1.REQ;
      E_CYCLE_1.EO TO Cons3.REQ;
      REAL2REAL_7_0_0.CNF TO F_MUL_6_0_0.REQ;
      REAL2REAL_2_2_1_0_0.CNF TO F_SUB_2_0.REQ;
      FB_INTEGRATE_1.CNF TO F_MUL_6_0.REQ;
      REAL2REAL_5_0_0.CNF TO F_SUB_3_0_0.REQ;
      F_ADD_2.CNF TO cons4.REQ;
      F_MUL_2_0.CNF TO REAL2REAL_2.REQ;
      F_SUB_5_0.CNF TO REAL2REAL_7_0_0.REQ;
      REAL2REAL_2_2_1_2.CNF TO F_DIV_3.REQ;
      F_ADD_2.CNF TO REAL2REAL_2_2_1_0.REQ;
      F_DIV_1.CNF TO mSC.REQ;
      REAL2REAL_5_0_0_0_0.CNF TO FB_INTEGRATE_1.REQ;
      REAL2REAL_7_0.CNF TO F_DIV_1.REQ;
      REAL2REAL_2.CNF TO F_MUL_2.REQ;
      F_MUL_2.CNF TO REAL2REAL_2_2_0.REQ;
      F_MUL_3_0.CNF TO REAL2REAL_5_0.REQ;
      F_SUB_3_0.CNF TO REAL2REAL_5_0_0.REQ;
      F_SUB_3_0_0.CNF TO REAL2REAL_5_0_0_0.REQ;
      m_air_inS.CNF TO m_air_inS_plus_noise.REQ;
      START.COLD TO FB_INTEGRATE_1.INIT;
      START.WARM TO FB_INTEGRATE_1.INIT;
      REAL2REAL_3_0.CNF TO F_SUB_5_0.REQ;
      mSC.CNF TO to_InputOutput2.REQ;
      FB_INTEGRATE_1.INITO TO to_InputOutput2.INIT;
      START.COLD TO from_EclipseScada1.INIT;
      START.WARM TO from_EclipseScada1.INIT;
      START.COLD TO from_EclipseScada6.INIT;
      START.WARM TO from_EclipseScada6.INIT;
      SUBSCRIBE_1_0.IND TO E_SWITCH.EI;
      E_SWITCH.EO1 TO E_CYCLE_1.START;
      START.COLD TO SUBSCRIBE_1_0.INIT;
      START.WARM TO SUBSCRIBE_1_0.INIT;
    END_CONNECTIONS
    DATA_CONNECTIONS
       TO ;
       TO ;
       TO ;
       TO ;
      mSB.OUT TO m_SB.IN;
      mCB.OUT TO m_CB.IN;
      mBG.OUT TO m_BG.IN;
      mGS.OUT TO m_GS.IN;
      mSC.OUT TO m_SC.IN;
      m_air_outS.OUT TO m_air_inC.IN;
      m_air_outS.OUT TO m_AirIN.IN;
      m_air_outS.OUT TO m_airS.IN;
      m_mois1.OUT TO m_mois.IN;
      mCFU.OUT TO m_CFU.IN;
      M_B2.OUT TO M_B.IN;
      M_G2.OUT TO M_G.IN;
      M_C2.OUT TO M_C.IN;
      m_air_outS.OUT TO m_airS1.IN;
      M_B2.OUT TO M_B1.IN;
      M_G2.OUT TO M_G1.IN;
      m_air_outS.OUT TO m_airS2.IN;
      M_S1.OUT TO M_S.IN;
      M_C2.OUT TO M_C1.IN;
      m_air_outS.OUT TO m_airS3.IN;
      M_G2.OUT TO M_G3.IN;
      Hg1.OUT TO Hg.IN;
      m_CB.OUT TO F_ADD_0.IN2;
      F_DIV.OUT TO mBG.IN;
      tauBG.OUT TO F_DIV.IN2;
      REAL2REAL_0_0.OUT TO F_ADD_0.IN1;
      FB_INTEGRATE.Y_OUT TO M_B2.IN;
      M_B2.OUT TO F_DIV.IN1;
      mBG.OUT TO F_SUB.IN2;
      REAL2REAL_0.OUT TO F_ADD.IN1;
      F_ADD.OUT TO REAL2REAL_0_0.IN;
      REAL2REAL_0_1_0.OUT TO FB_INTEGRATE.X;
      m_SB.OUT TO F_ADD.IN2;
      F_MUL.OUT TO REAL2REAL_0.IN;
      REAL2REAL_0_1.OUT TO F_SUB.IN1;
      a1.OUT TO F_MUL.IN2;
      F_ADD_0.OUT TO REAL2REAL_0_1.IN;
      F_SUB.OUT TO REAL2REAL_0_1_0.IN;
      mF.OUT TO F_MUL.IN1;
      MV_from_ESCADA.RD_1 TO mF.IN;
      PP_from_ESCADA1.RD_1 TO a1.IN;
      PP_from_ESCADA1.RD_2 TO tauBG.IN;
      START_Subscribe.RD_1 TO E_SWITCH_0.G;
      gamma1.OUT TO F_MUL_1.IN1;
      REAL2REAL_2_0_0.OUT TO FB_INTEGRATE_0.X;
      mGS.OUT TO F_SUB_0.IN2;
      REAL2REAL_2_0_3.OUT TO F_MUL_1_3.IN1;
      F_MUL_1_2.OUT TO REAL2REAL_2_0_3.IN;
      bJ.OUT TO F_MUL_1_2.IN1;
      gammaJ.OUT TO F_MUL_1_3.IN2;
      REAL2REAL_2_0_3_0_0.OUT TO F_ADD_1.IN2;
      tauGS.OUT TO F_DIV_0.IN2;
      FB_INTEGRATE_0.Y_OUT TO F_MUL_1.IN2;
      F_SUB_0_0.OUT TO REAL2REAL_2_0_3_0_0.IN;
      REAL2REAL_2_0_3_0.OUT TO F_SUB_0_0.IN2;
      F_SUB_0.OUT TO REAL2REAL_2_0_0.IN;
      REAL2REAL_2_0.OUT TO F_SUB_0.IN1;
      FB_INTEGRATE_0.Y_OUT TO M_G2.IN;
      FB_INTEGRATE_0.Y_OUT TO F_DIV_0.IN1;
      m_BG.OUT TO F_ADD_1.IN1;
      F_DIV_0.OUT TO mGS.IN;
      F_MUL_1_3.OUT TO REAL2REAL_2_0_3_1.IN;
      F_ADD_1.OUT TO REAL2REAL_2_0.IN;
      REAL2REAL_2_0_3_1.OUT TO F_SUB_0_0.IN1;
      F_MUL_1.OUT TO REAL2REAL_2_0_3_0.IN;
      FB_INTEGRATE_0.Y_OUT TO F_MUL_1_2.IN2;
      M_G2.OUT TO to_InputOutput1.SD_1;
      mGS.OUT TO to_InputOutput1.SD_2;
      from_EclipseScada5.RD_1 TO gamma1.IN;
      from_EclipseScada5.RD_2 TO bJ.IN;
      from_EclipseScada5.RD_3 TO gammaJ.IN;
      from_EclipseScada5.RD_4 TO tauGS.IN;
      SUBSCRIBE_1_2.RD_1 TO E_SWITCH_1.G;
      m_SC.OUT TO F_ADD_3_0.IN1;
      Cons1_0.OUT TO F_MUL_2_1.IN1;
      REAL2REAL_8_0.OUT TO F_SUB_4_0_0.IN1;
      REAL2REAL_21.OUT TO F_SUB_4_0.IN1;
      Cons3_0.OUT TO F_ADD_2_0.IN2;
      d_max_0.OUT TO F_SUB_2_0_0.IN1;
      tau_CB.OUT TO F_DIV_5_0.IN2;
      REAL2REAL_2_2_1_0_0_0.OUT TO F_SUB_2_1.IN1;
      REAL2REAL_2_2_0_1_0.OUT TO F_ADD_2_0.IN1;
      m_air_inC.OUT TO m_air_outC.IN;
      F_SUB_2_0_0.OUT TO REAL2REAL_2_2_1_1_0.IN;
      F_DIV_5_0.OUT TO mCB.IN;
      F_MUL_5_0.OUT TO REAL2REAL_2_2_1_0_0_0.IN;
      d_min_0.OUT TO F_SUB_2_1.IN2;
      REAL2REAL_10_0.OUT TO F_DIV_5.IN1;
      m_air_inC.OUT TO F_MUL_2_0_1.IN2;
      m_air_inC.OUT TO F_MUL_2_0_1.IN1;
      F_ADD_3_0.OUT TO REAL2REAL_21.IN;
      d_min_0.OUT TO F_SUB_2_0_0.IN2;
      REAL2REAL_10_0_0_0.OUT TO F_MUL_7_0.IN1;
      F_SUB_2_1.OUT TO REAL2REAL_2_2_1_2_0.IN;
      m_air_inC.OUT TO F_MUL_2_0_0_0.IN1;
      FB_INTEGRATE_2.Y_OUT TO M_C2.IN;
      F_SUB_4_0.OUT TO REAL2REAL_8_0.IN;
      REAL2REAL_10_0_0.OUT TO F_SUB_7_0.IN1;
      F_MUL_7.OUT TO REAL2REAL_10_0.IN;
      F_MUL_7_0.OUT TO REAL2REAL_10_1.IN;
      REAL2REAL_2_2_1.OUT TO F_SUB_1_0.IN2;
      F_MUL_2_0_0_0.OUT TO REAL2REAL_2_2_1.IN;
      F_DIV_4.OUT TO c2.IN;
      c2.OUT TO F_MUL_7.IN2;
      F_MUL_2_1.OUT TO REAL2REAL_2_2_0_0.IN;
      F_SUB_4_0_0.OUT TO REAL2REAL_8_0_0.IN;
      REAL2REAL_2_2_0_0.OUT TO F_SUB_1_0.IN1;
      F_MUL_2_0_1.OUT TO REAL2REAL_2_1.IN;
      REAL2REAL_8_0_0.OUT TO FB_INTEGRATE_2.X;
      FB_INTEGRATE_2.Y_OUT TO F_MUL_7.IN1;
      mCFU.OUT TO F_SUB_4_0.IN2;
      F_SUB_7_0.OUT TO REAL2REAL_10_0_0_0.IN;
      REAL2REAL_10_1.OUT TO F_DIV_5_0.IN1;
      c2.OUT TO F_SUB_7_0.IN2;
      cons4_0.OUT TO F_MUL_5_0.IN2;
      F_ADD_2_0.OUT TO REAL2REAL_2_2_1_0_1.IN;
      REAL2REAL_2_2_1_0_1.OUT TO F_MUL_5_0.IN1;
      REAL2REAL_2_2_1_2_0.OUT TO F_DIV_4.IN1;
      F_SUB_1_0.OUT TO REAL2REAL_2_2_0_1_0.IN;
      FB_INTEGRATE_2.Y_OUT TO F_MUL_7_0.IN2;
      REAL2REAL_2_2_1_1_0.OUT TO F_DIV_4.IN2;
      mCB.OUT TO F_SUB_4_0_0.IN2;
      F_DIV_5.OUT TO mCFU.IN;
      Cons2_0.OUT TO F_MUL_2_0_0_0.IN2;
      m_AirIN.OUT TO F_ADD_3_0.IN2;
      REAL2REAL_2_1.OUT TO F_MUL_2_1.IN2;
      tau_CFU.OUT TO F_DIV_5.IN2;
      M_C2.OUT TO to_InputOutput3.SD_1;
      mCB.OUT TO to_InputOutput3.SD_2;
      mCFU.OUT TO to_InputOutput3.SD_3;
      m_air_outC.OUT TO to_InputOutput3.SD_4;
      SUBSCRIBE_1_3.RD_1 TO E_SWITCH_2.G;
      from_EclipseScada7.RD_1 TO d_min_0.IN;
      from_EclipseScada7.RD_2 TO d_max_0.IN;
      from_EclipseScada7.RD_3 TO tau_CB.IN;
      from_EclipseScada7.RD_4 TO tau_CFU.IN;
      REAL2REAL_33_0.OUT TO F_ADD_8.IN2;
      REAL2REAL_37_0.OUT TO F_DIV_6.IN1;
      F_MUL_9.OUT TO REAL2REAL_9_0.IN;
      REAL2REAL_16_0.OUT TO F_MUL_17.IN1;
      M_met.OUT TO F_MUL_26_0.IN1;
      REAL2REAL_48_0.OUT TO F_ADD_15.IN1;
      theta_FB.OUT TO F_MUL_12.IN2;
      F_MUL_21_0.OUT TO REAL2REAL_30_0.IN;
      Cp_w.OUT TO F_MUL_13.IN1;
      F_ADD_9.OUT TO REAL2REAL_36_0.IN;
      REAL2REAL_46_0.OUT TO F_MUL_30_0.IN1;
      F_ADD_4.OUT TO REAL2REAL_19_0.IN;
      F_MUL_13.OUT TO REAL2REAL_14_0.IN;
      REAL2REAL_49_0.OUT TO F_DIV_6.IN2;
      T_a.OUT TO F_MUL_10.IN2;
      F_ADD_7.OUT TO REAL2REAL_23_0.IN;
      m_CF.OUT TO F_MUL_12.IN1;
      F_MUL_11.OUT TO REAL2REAL_12_0.IN;
      F_MUL_25_0.OUT TO REAL2REAL_32_0.IN;
      F_ADD_15.OUT TO REAL2REAL_49_0.IN;
      Cp_c.OUT TO F_MUL_18_0.IN1;
      F_ADD_10.OUT TO REAL2REAL_39_0.IN;
      REAL2REAL_40_0.OUT TO F_MUL_27_0.IN1;
      theta_acc.OUT TO F_SUB_12.IN2;
      T_out.OUT TO F_MUL_21_0.IN2;
      K_loss.OUT TO F_MUL_15_0.IN1;
      REAL2REAL_22_0.OUT TO F_ADD_7.IN2;
      REAL2REAL_35_0.OUT TO F_ADD_9.IN2;
      Satu.OUT TO F_SUB_6.IN1;
      theta_out.OUT TO F_SUB_9.IN2;
      REAL2REAL_42_0.OUT TO F_MUL_28_0.IN1;
      theta_FB.OUT TO F_SUB_6.IN2;
      Cp_a.OUT TO F_MUL_0.IN2;
      m_mois.OUT TO F_MUL_13_0.IN1;
      REAL2REAL_47_0.OUT TO F_ADD_15.IN2;
      F_MUL_14.OUT TO REAL2REAL_15_0.IN;
      REAL2REAL_19_0.OUT TO F_ADD_7.IN1;
      F_ADD_6.OUT TO REAL2REAL_22_0.IN;
      F_MUL_26_0.OUT TO REAL2REAL_38_0.IN;
      F_MUL_0.OUT TO REAL2REAL_1_0.IN;
      T_a.OUT TO F_MUL_15_0.IN2;
      m_CFU.OUT TO F_MUL_16_0.IN1;
      F_SUB_12.OUT TO REAL2REAL_41_0.IN;
      REAL2REAL_14_0.OUT TO F_MUL_14.IN2;
      theta_acc.OUT TO F_MUL_29_0.IN2;
      REAL2REAL_29_0.OUT TO F_MUL_22_0.IN1;
      REAL2REAL_32_0.OUT TO F_ADD_8.IN1;
      F_MUL_10.OUT TO REAL2REAL_11_0.IN;
      M_B.OUT TO F_ADD_12.IN1;
      dT_out.OUT TO FB_INTEGRATE_3.X;
      REAL2REAL_12_0.OUT TO F_ADD_4.IN2;
      F_MUL_16_0.OUT TO REAL2REAL_25_0.IN;
      M_G.OUT TO F_ADD_10.IN2;
      REAL2REAL_15_0.OUT TO F_ADD_5.IN1;
      F_MUL_24_0.OUT TO REAL2REAL_28_0.IN;
      Cp_c1.OUT TO F_MUL_28_0.IN2;
      Hg.OUT TO F_ADD_5.IN2;
      Cp1.OUT TO F_MUL_24_0.IN2;
      Satu1.OUT TO F_SUB_9.IN1;
      F_MUL_13_0.OUT TO REAL2REAL_16_0.IN;
      REAL2REAL_25_0.OUT TO F_MUL_19_0.IN1;
      M_C.OUT TO F_ADD_13.IN2;
      Satu2.OUT TO F_SUB_12.IN1;
      T_m_air.OUT TO F_MUL_8.IN2;
      REAL2REAL_13_0.OUT TO F_MUL_14.IN1;
      F_MUL_18_0.OUT TO REAL2REAL_26_0.IN;
      Cp.OUT TO F_MUL_10.IN1;
      F_DIV_6.OUT TO dT_out.IN;
      F_MUL_17.OUT TO REAL2REAL_17_0.IN;
      REAL2REAL_1_0.OUT TO F_MUL_8.IN1;
      F_MUL_12.OUT TO REAL2REAL_13_0.IN;
      F_MUL_20_0.OUT TO REAL2REAL_29_0.IN;
      F_ADD_8.OUT TO REAL2REAL_35_0.IN;
      REAL2REAL_44_0.OUT TO F_ADD_13.IN1;
      F_MUL_29_0.OUT TO REAL2REAL_46_0.IN;
      M_G.OUT TO F_ADD_12.IN2;
      F_SUB_6.OUT TO REAL2REAL_6_0.IN;
      REAL2REAL_28_0.OUT TO F_MUL_25_0.IN1;
      h.OUT TO F_MUL_13_0.IN2;
      REAL2REAL_26_0.OUT TO F_MUL_19_0.IN2;
      F_ADD_13.OUT TO REAL2REAL_45_0.IN;
      REAL2REAL_34_0.OUT TO F_ADD_9.IN1;
      v_t.OUT TO F_MUL_17.IN2;
      F_SUB_8.OUT TO REAL2REAL_21_0.IN;
      F_ADD_11.OUT TO REAL2REAL_40_0.IN;
      T_out.OUT TO F_MUL_23_0.IN2;
      F_SUB_9.OUT TO REAL2REAL_24_0.IN;
      REAL2REAL_4_0.OUT TO F_ADD_4.IN1;
      F_MUL_22_0.OUT TO REAL2REAL_31_0.IN;
      REAL2REAL_21_0.OUT TO F_ADD_6.IN2;
      F_MUL_30_0.OUT TO REAL2REAL_47_0.IN;
      F_MUL_28_0.OUT TO REAL2REAL_43_0.IN;
      REAL2REAL_9_0.OUT TO F_MUL_11.IN1;
      F_MUL_23_0.OUT TO REAL2REAL_33_0.IN;
      M_C.OUT TO F_ADD_11.IN2;
      REAL2REAL_45_0.OUT TO F_MUL_29_0.IN1;
      REAL2REAL_20_0.OUT TO F_ADD_6.IN1;
      Cp_w1.OUT TO F_MUL_21_0.IN1;
      Cp_met.OUT TO F_MUL_26_0.IN2;
      M_B.OUT TO F_ADD_10.IN1;
      REAL2REAL_30_0.OUT TO F_MUL_22_0.IN2;
      REAL2REAL_24_0.OUT TO F_MUL_16_0.IN2;
      F_MUL_15_0.OUT TO REAL2REAL_18_0.IN;
      REAL2REAL_36_0.OUT TO F_SUB_11.IN2;
      m_CF.OUT TO F_MUL_9.IN1;
      F_MUL_27_0.OUT TO REAL2REAL_42_0.IN;
      Cp_w2.OUT TO F_MUL_30_0.IN2;
      REAL2REAL_11_0.OUT TO F_MUL_11.IN2;
      m_CFU.OUT TO F_MUL_20_0.IN1;
      m_airS.OUT TO F_MUL_0.IN1;
      REAL2REAL_39_0.OUT TO F_ADD_11.IN1;
      T_out.OUT TO F_MUL_18_0.IN2;
      F_SUB_11.OUT TO REAL2REAL_37_0.IN;
      REAL2REAL_41_0.OUT TO F_MUL_27_0.IN2;
      FB_INTEGRATE_3.Y_OUT TO T_out.IN;
      REAL2REAL_38_0.OUT TO F_ADD_14.IN1;
      F_MUL_8.OUT TO REAL2REAL_4_0.IN;
      T_a.OUT TO F_MUL_13.IN2;
      F_ADD_12.OUT TO REAL2REAL_44_0.IN;
      REAL2REAL_6_0.OUT TO F_MUL_9.IN2;
      m_airS.OUT TO F_MUL_24_0.IN1;
      F_MUL_19_0.OUT TO REAL2REAL_27_0.IN;
      REAL2REAL_43_0.OUT TO F_ADD_14.IN2;
      REAL2REAL_23_0.OUT TO F_SUB_11.IN1;
      T_out.OUT TO F_MUL_25_0.IN2;
      F_ADD_5.OUT TO REAL2REAL_20_0.IN;
      F_ADD_14.OUT TO REAL2REAL_48_0.IN;
      K_loss1.OUT TO F_MUL_23_0.IN1;
      theta_out.OUT TO F_MUL_20_0.IN2;
      T_out.OUT TO to_InputOutput4.SD_1;
      from_EclipseScada2.RD_1 TO T_m_air.IN;
      from_EclipseScada2.RD_2 TO m_CF.IN;
      from_EclipseScada2.RD_3 TO T_a.IN;
      from_EclipseScada2.RD_4 TO M_met.IN;
      SUBSCRIBE_1_4.RD_1 TO E_SWITCH_3.G;
      from_EclipseScada8.RD_1 TO Cp_a.IN;
      from_EclipseScada8.RD_2 TO theta_FB.IN;
      from_EclipseScada8.RD_3 TO Cp.IN;
      from_EclipseScada8.RD_4 TO Cp_w.IN;
      from_EclipseScada8.RD_5 TO h.IN;
      from_EclipseScada8.RD_6 TO v_t.IN;
      from_EclipseScada9.RD_1 TO K_loss.IN;
      from_EclipseScada9.RD_2 TO theta_out.IN;
      from_EclipseScada9.RD_3 TO Cp_c.IN;
      from_EclipseScada9.RD_4 TO Cp_w1.IN;
      from_EclipseScada9.RD_5 TO Cp1.IN;
      from_EclipseScada9.RD_6 TO K_loss1.IN;
      from_EclipseScada10.RD_1 TO Cp_met.IN;
      from_EclipseScada10.RD_2 TO theta_acc.IN;
      from_EclipseScada10.RD_3 TO Cp_c1.IN;
      from_EclipseScada10.RD_4 TO Cp_w2.IN;
      REAL2REAL_17_0.OUT TO F_SUB_8.IN2;
      REAL2REAL_18_0.OUT TO F_SUB_8.IN1;
      REAL2REAL_27_0.OUT TO F_ADD_3.IN1;
      REAL2REAL_31_0.OUT TO F_ADD_3.IN2;
      F_ADD_3.OUT TO REAL2REAL_34_0.IN;
      M_S.OUT TO F_ADD_17.IN1;
      F_ADD_17.OUT TO REAL2REAL_59.IN;
      F_MUL_32.OUT TO REAL2REAL_53.IN;
      m_airS2.OUT TO F_MUL_33.IN2;
      REAL2REAL_60.OUT TO F_MUL_38.IN1;
      m_airS2.OUT TO F_MUL_33.IN1;
      REAL2REAL_53.OUT TO F_ADD_18.IN1;
      F_MUL_31.OUT TO REAL2REAL_52.IN;
      F_ADD_16.OUT TO REAL2REAL_54.IN;
      F_ADD_18.OUT TO REAL2REAL_62.IN;
      K_ce.OUT TO F_MUL_37.IN1;
      REAL2REAL_56.OUT TO F_MUL_35.IN1;
      m_airS3.OUT TO F_MUL_36.IN1;
      m_airS3.OUT TO F_MUL_36.IN2;
      REAL2REAL_52.OUT TO F_MUL_32.IN2;
      REAL2REAL_54.OUT TO F_MUL_34.IN2;
      REAL2REAL_55.OUT TO F_MUL_35.IN2;
      REAL2REAL_58.OUT TO F_MUL_38.IN2;
      M_G1.OUT TO F_ADD_16.IN2;
      F_ADD_19.OUT TO dP_mill.IN;
      REAL2REAL_59.OUT TO F_MUL_37.IN2;
      K_c.OUT TO F_MUL_34.IN1;
      F_MUL_37.OUT TO REAL2REAL_60.IN;
      REAL2REAL_62.OUT TO F_ADD_19.IN1;
      F_MUL_34.OUT TO REAL2REAL_56.IN;
      REAL2REAL_57.OUT TO F_ADD_18.IN2;
      m_airS1.OUT TO F_MUL_31.IN1;
      REAL2REAL_61.OUT TO F_ADD_19.IN2;
      m_airS1.OUT TO F_MUL_31.IN2;
      M_B1.OUT TO F_ADD_16.IN1;
      F_MUL_38.OUT TO REAL2REAL_61.IN;
      F_MUL_35.OUT TO REAL2REAL_57.IN;
      M_C1.OUT TO F_ADD_17.IN2;
      F_MUL_36.OUT TO REAL2REAL_58.IN;
      F_MUL_33.OUT TO REAL2REAL_55.IN;
      K_auf.OUT TO F_MUL_32.IN1;
      dP_mill.OUT TO to_InputOutput5.SD_1;
      SUBSCRIBE_1_5.RD_1 TO E_SWITCH_4.G;
      from_EclipseScada11.RD_1 TO K_auf.IN;
      from_EclipseScada11.RD_2 TO K_c.IN;
      from_EclipseScada11.RD_3 TO K_ce.IN;
      F_MUL_40.OUT TO REAL2REAL_51.IN;
      F_MUL_43.OUT TO REAL2REAL_66.IN;
      P_load.OUT TO F_ADD_20.IN2;
      F_DIV_7.OUT TO I_total.IN;
      REAL2REAL_63.OUT TO F_ADD_20.IN1;
      REAL2REAL_50.OUT TO F_MUL_41.IN1;
      M_on.OUT TO F_MUL_42.IN2;
      P_f.OUT TO F_MUL_43.IN2;
      K_power.OUT TO F_MUL_39.IN1;
      w.OUT TO F_MUL_40.IN1;
      N_rol.OUT TO F_MUL_40.IN2;
      I_total.OUT TO F_MUL_44.IN1;
      F_ADD_20.OUT TO REAL2REAL_64.IN;
      P_total.OUT TO F_DIV_7.IN1;
      M_G3.OUT TO F_MUL_39.IN2;
      F_MUL_41.OUT TO REAL2REAL_63.IN;
      M_v.OUT TO F_MUL_43.IN1;
      F_MUL_39.OUT TO REAL2REAL_50.IN;
      REAL2REAL_66.OUT TO F_DIV_7.IN2;
      F_MUL_42.OUT TO P_total.IN;
      REAL2REAL_64.OUT TO F_MUL_42.IN1;
      REAL2REAL_51.OUT TO F_MUL_41.IN2;
      F_MUL_44.OUT TO Hg1.IN;
      K_g.OUT TO F_MUL_44.IN2;
      P_total.OUT TO to_InputOutput6.SD_1;
      I_total.OUT TO to_InputOutput6.SD_2;
      Hg1.OUT TO to_InputOutput6.SD_3;
      from_EclipseScada3.RD_1 TO P_load.IN;
      SUBSCRIBE_1_6.RD_1 TO E_SWITCH_5.G;
      from_EclipseScada12.RD_1 TO K_power.IN;
      from_EclipseScada12.RD_2 TO w.IN;
      from_EclipseScada12.RD_3 TO N_rol.IN;
      from_EclipseScada12.RD_4 TO M_on.IN;
      from_EclipseScada13.RD_1 TO M_v.IN;
      from_EclipseScada13.RD_2 TO P_f.IN;
      from_EclipseScada13.RD_3 TO K_g.IN;
      REAL2REAL_7_0.OUT TO F_DIV_1.IN1;
      F_SUB_3_0_0.OUT TO REAL2REAL_5_0_0_0.IN;
      tauSB.OUT TO F_DIV_2.IN2;
      nu_acc.OUT TO F_MUL_3_0.IN2;
      REAL2REAL_2_2_0_1.OUT TO F_ADD_2.IN1;
      F_MUL_4_0.OUT TO m_mois1.IN;
      REAL2REAL_2_2_1_1.OUT TO F_DIV_3.IN2;
      F_MUL_6_0.OUT TO REAL2REAL_7_0.IN;
      c1.OUT TO F_SUB_5_0.IN2;
      FB_INTEGRATE_1.Y_OUT TO M_S1.IN;
      F_MUL_2.OUT TO REAL2REAL_2_2_0.IN;
      Cons2.OUT TO F_MUL_2_0_0.IN2;
      tauSC.OUT TO F_DIV_1.IN2;
      REAL2REAL_2_2_1_0_0.OUT TO F_SUB_2.IN1;
      m_GS.OUT TO F_MUL_4_0.IN2;
      REAL2REAL_5_0_0_0_0.OUT TO FB_INTEGRATE_1.X;
      F_SUB_3_0_0_0.OUT TO REAL2REAL_5_0_0_0_0.IN;
      F_SUB_1.OUT TO REAL2REAL_2_2_0_1.IN;
      F_MUL_6_0_0.OUT TO REAL2REAL_7_1.IN;
      mSB.OUT TO F_SUB_3_0_0.IN2;
      m_mois1.OUT TO F_SUB_3_0.IN2;
      FB_INTEGRATE_1.Y_OUT TO F_MUL_6_0_0.IN2;
      m_air_inS_plus_noise.OUT TO F_MUL_2_0_0.IN1;
      FB_INTEGRATE_1.Y_OUT TO F_MUL_6_0.IN2;
      d_min.OUT TO F_SUB_2.IN2;
      m_GS.OUT TO F_SUB_3_0.IN1;
      Cons3.OUT TO F_ADD_2.IN2;
      F_DIV_3.OUT TO c1.IN;
      rho.OUT TO F_MUL_3_0.IN1;
      c1.OUT TO F_MUL_6_0.IN1;
      REAL2REAL_3_0.OUT TO F_SUB_5_0.IN1;
      F_ADD_2.OUT TO REAL2REAL_2_2_1_0.IN;
      Cons1.OUT TO F_MUL_2.IN1;
      F_MUL_3_0.OUT TO REAL2REAL_5_0.IN;
      REAL2REAL_7_1.OUT TO F_DIV_2.IN1;
      d_min.OUT TO F_SUB_2_0.IN2;
      REAL2REAL_2_2.OUT TO F_SUB_1.IN2;
      F_SUB_2_0.OUT TO REAL2REAL_2_2_1_1.IN;
      cons4.OUT TO F_MUL_5.IN2;
      F_MUL_5.OUT TO REAL2REAL_2_2_1_0_0.IN;
      REAL2REAL_5_0_0.OUT TO F_SUB_3_0_0.IN1;
      REAL2REAL_2_2_0.OUT TO F_SUB_1.IN1;
      F_SUB_5_0.OUT TO REAL2REAL_7_0_0.IN;
      REAL2REAL_7_0_0.OUT TO F_MUL_6_0_0.IN1;
      F_DIV_1.OUT TO mSC.IN;
      REAL2REAL_5_0.OUT TO F_MUL_4_0.IN1;
      d_max.OUT TO F_SUB_2_0.IN1;
      REAL2REAL_2_2_1_2.OUT TO F_DIV_3.IN1;
      m_air_inS_plus_noise.OUT TO m_air_outS.IN;
      m_air_inS_plus_noise.OUT TO F_MUL_2_0.IN1;
      m_air_inS_plus_noise.OUT TO F_MUL_2_0.IN2;
      F_MUL_2_0_0.OUT TO REAL2REAL_2_2.IN;
      mSC.OUT TO F_SUB_3_0_0_0.IN2;
      F_SUB_3_0.OUT TO REAL2REAL_5_0_0.IN;
      REAL2REAL_2.OUT TO F_MUL_2.IN2;
      REAL2REAL_5_0_0_0.OUT TO F_SUB_3_0_0_0.IN1;
      F_DIV_2.OUT TO mSB.IN;
      F_SUB_2.OUT TO REAL2REAL_2_2_1_2.IN;
      F_MUL_2_0.OUT TO REAL2REAL_2.IN;
      REAL2REAL_2_2_1_0.OUT TO F_MUL_5.IN1;
      m_air_inS.OUT TO m_air_inS_plus_noise.IN;
      M_S1.OUT TO to_InputOutput2.SD_1;
      mSC.OUT TO to_InputOutput2.SD_2;
      m_air_outS.OUT TO to_InputOutput2.SD_3;
      mSB.OUT TO to_InputOutput2.SD_4;
      m_mois1.OUT TO to_InputOutput2.SD_5;
      from_EclipseScada1.RD_1 TO m_air_inS.IN;
      from_EclipseScada6.RD_1 TO d_min.IN;
      from_EclipseScada6.RD_2 TO d_max.IN;
      from_EclipseScada6.RD_3 TO rho.IN;
      from_EclipseScada6.RD_4 TO nu_acc.IN;
      from_EclipseScada6.RD_5 TO tauSB.IN;
      from_EclipseScada6.RD_6 TO tauSC.IN;
      SUBSCRIBE_1_0.RD_1 TO E_SWITCH.G;
    END_CONNECTIONS
  END_APPLICATION
  APPLICATION InputOutput
    FBS
      from_GrindingZone : SUBSCRIBE_2(QI := 1, ID := 127.0.0.1:62200);
      to_ESCADA2 : PUBLISH_1(QI := 1, ID := sfp[ProcessVariable.GrindingZone.M_G]);
      REAL2REAL_69 : REAL2REAL;
      REAL2REAL_68 : REAL2REAL;
      to_ESCADA3 : PUBLISH_1(QI := 1, ID := sfp[ProcessVariable.GrindingZone.m_GS]);
      to_ESCADA8 : PUBLISH_1(QI := 1, ID := sfp[ProcessVariable.SeparatorZone.m_moiss]);
      REAL2REAL_72 : REAL2REAL;
      to_ESCADA4 : PUBLISH_1(QI := 1, ID := sfp[ProcessVariable.SeparatorZone.M_S]);
      to_ESCADA7 : PUBLISH_1(QI := 1, ID := sfp[ProcessVariable.SeparatorZone.m_SB]);
      from_SeparatorZone : SUBSCRIBE_5(QI := 1, ID := 127.0.0.1:62300);
      REAL2REAL_70 : REAL2REAL;
      to_ESCADA6 : PUBLISH_1(QI := 1, ID := sfp[ProcessVariable.SeparatorZone.m_air_outS]);
      to_ESCADA5 : PUBLISH_1(QI := 1, ID := sfp[ProcessVariable.SeparatorZone.m_SC]);
      REAL2REAL_74 : REAL2REAL;
      REAL2REAL_71 : REAL2REAL;
      REAL2REAL_73 : REAL2REAL;
      REAL2REAL_75 : REAL2REAL;
      tp_ESCADA10 : PUBLISH_1(QI := 1, ID := sfp[ProcessVariable.ClassifierZone.m_CB]);
      to_ESCADA9 : PUBLISH_1(QI := 1, ID := sfp[ProcessVariable.ClassifierZone.M_C]);
      REAL2REAL_77 : REAL2REAL;
      REAL2REAL_78 : REAL2REAL;
      to_ESCADA12 : PUBLISH_1(QI := 1, ID := sfp[ProcessVariable.ClassifierZone.m_air_outC]);
      to_ESCADA11 : PUBLISH_1(QI := 1, ID := sfp[ProcessVariable.ClassifierZone.m_CFU]);
      from_ClassifierZone : SUBSCRIBE_4(QI := 1, ID := 127.0.0.1:62400);
      REAL2REAL_76 : REAL2REAL;
      REAL2REAL_79 : REAL2REAL;
      to_ESCADA13 : PUBLISH_1(QI := 1, ID := sfp[ProcessVariable.HeatBalances.T_out]);
      from_HeatBalances : SUBSCRIBE_1(QI := 1, ID := 127.0.0.1:62500);
      REAL2REAL_80 : REAL2REAL;
      from_DifferentialPressureBalances : SUBSCRIBE_1(QI := 1, ID := 127.0.0.1:62600);
      to_ESCADA14 : PUBLISH_1(QI := 1, ID := sfp[ProcessVariable.DifferentialPressureBalances.dP_mill]);
      to_ESCADA16 : PUBLISH_1(QI := 1, ID := sfp[ProcessVariable.PowerBalances.I_total]);
      REAL2REAL_82 : REAL2REAL;
      REAL2REAL_83 : REAL2REAL;
      to_ESCADA15 : PUBLISH_1(QI := 1, ID := sfp[ProcessVariable.PowerBalances.P_total]);
      REAL2REAL_81 : REAL2REAL;
      to_ESCADA17 : PUBLISH_1(QI := 1, ID := sfp[ProcessVariable.PowerBalances.Hg]);
      from_PowerBalances : SUBSCRIBE_3(QI := 1, ID := 127.0.0.1:62700);
      to_BowlZone : PUBLISH_1(QI := 1, ID := 127.0.0.1:63100);
      m_F : REAL2REAL;
      from_ESCADA : SUBSCRIBE_1(QI := 1, ID := sfp[ManipulatedVariable.BowlZone.m_F]);
      from_ESCADA1 : SUBSCRIBE_1(QI := 1, ID := sfp[ManipulatedVariable.SeparatorZone.m_air_inS]);
      to_SeparatorZone : PUBLISH_1(QI := 1, ID := 127.0.0.1:63300);
      REAL2REAL_85 : REAL2REAL;
      REAL2REAL_89 : REAL2REAL;
      REAL2REAL_88 : REAL2REAL;
      from_ESCADA4 : SUBSCRIBE_1(QI := 1, ID := sfp[ManipulatedVariable.HeatBalances.T_a]);
      from_ESCADA5 : SUBSCRIBE_1(QI := 1, ID := sfp[ManipulatedVariable.HeatBalances.M_met]);
      REAL2REAL_86 : REAL2REAL;
      from_ESCADA2 : SUBSCRIBE_1(QI := 1, ID := sfp[ManipulatedVariable.HeatBalances.T_m_air]);
      to_HeatBalances : PUBLISH_4(QI := 1, ID := 127.0.0.1:63500);
      from_ESCADA3 : SUBSCRIBE_1(QI := 1, ID := sfp[ManipulatedVariable.HeatBalances.m_CF]);
      REAL2REAL_87 : REAL2REAL;
      from_ESCADA6 : SUBSCRIBE_1(QI := 1, ID := sfp[ManipulatedVariable.PowerBalances.P_load]);
      REAL2REAL_90 : REAL2REAL;
      to_PowerBalances : PUBLISH_1(QI := 1, ID := 127.0.0.1:63700);
      a_i : REAL2REAL;
      t_BG : REAL2REAL;
      from_ESCADA8 : SUBSCRIBE_1(QI := 1, ID := sfp[ProcessParameter.BowlZone.t_BG]);
      to_BowlZone2 : PUBLISH_2(QI := 1, ID := 127.0.0.1:64100);
      from_ESCADA7 : SUBSCRIBE_1(QI := 1, ID := sfp[ProcessParameter.BowlZone.a_i]);
      from_ESCADA10 : SUBSCRIBE_1(QI := 1, ID := sfp[ProcessParameter.GrindingZone.b_J]);
      from_ESCADA11 : SUBSCRIBE_1(QI := 1, ID := sfp[ProcessParameter.GrindingZone.gamma_J]);
      REAL2REAL_93 : REAL2REAL;
      to_GrindingZone : PUBLISH_4(QI := 1, ID := 127.0.0.1:64200);
      REAL2REAL_95 : REAL2REAL;
      REAL2REAL_94 : REAL2REAL;
      from_ESCADA12 : SUBSCRIBE_1(QI := 1, ID := sfp[ProcessParameter.GrindingZone.t_GS]);
      from_ESCADA9 : SUBSCRIBE_1(QI := 1, ID := sfp[ProcessParameter.GrindingZone.gamma_i]);
      REAL2REAL_96 : REAL2REAL;
      REAL2REAL_98 : REAL2REAL;
      REAL2REAL_102 : REAL2REAL;
      REAL2REAL_97 : REAL2REAL;
      from_ESCADA16 : SUBSCRIBE_1(QI := 1, ID := sfp[ProcessParameter.SeparatorZone.nu_acc]);
      REAL2REAL_99 : REAL2REAL;
      REAL2REAL_100 : REAL2REAL;
      from_ESCADA15 : SUBSCRIBE_1(QI := 1, ID := sfp[ProcessParameter.SeparatorZone.rho]);
      from_ESCADA14 : SUBSCRIBE_1(QI := 1, ID := sfp[ProcessParameter.SeparatorZone.d_max]);
      to_SeparatorZone1 : PUBLISH_6(QI := 1, ID := 127.0.0.1:64300);
      from_ESCADA17 : SUBSCRIBE_1(QI := 1, ID := sfp[ProcessParameter.SeparatorZone.t_SB]);
      REAL2REAL_101 : REAL2REAL;
      from_ESCADA18 : SUBSCRIBE_1(QI := 1, ID := sfp[ProcessParameter.SeparatorZone.t_SC]);
      from_ESCADA13 : SUBSCRIBE_1(QI := 1, ID := sfp[ProcessParameter.SeparatorZone.d_min]);
      from_ESCADA22 : SUBSCRIBE_1(QI := 1, ID := sfp[ProcessParameter.ClassifierZone.t_CFU]);
      REAL2REAL_104 : REAL2REAL;
      to_ClassifierZone : PUBLISH_4(QI := 1, ID := 127.0.0.1:64400);
      from_ESCADA20 : SUBSCRIBE_1(QI := 1, ID := sfp[ProcessParameter.ClassifierZone.d_max]);
      REAL2REAL_106 : REAL2REAL;
      from_ESCADA19 : SUBSCRIBE_1(QI := 1, ID := sfp[ProcessParameter.ClassifierZone.d_min]);
      REAL2REAL_103 : REAL2REAL;
      from_ESCADA21 : SUBSCRIBE_1(QI := 1, ID := sfp[ProcessParameter.ClassifierZone.t_CB]);
      REAL2REAL_105 : REAL2REAL;
      REAL2REAL_108 : REAL2REAL;
      REAL2REAL_110 : REAL2REAL;
      from_ESCADA26 : SUBSCRIBE_1(QI := 1, ID := sfp[ProcessParameter.HeatBalances.Cp_w]);
      from_ESCADA24 : SUBSCRIBE_1(QI := 1, ID := sfp[ProcessParameter.HeatBalances.theta_FB]);
      from_ESCADA23 : SUBSCRIBE_1(QI := 1, ID := sfp[ProcessParameter.HeatBalances.Cp_a]);
      from_ESCADA25 : SUBSCRIBE_1(QI := 1, ID := sfp[ProcessParameter.HeatBalances.Cp]);
      from_ESCADA28 : SUBSCRIBE_1(QI := 1, ID := sfp[ProcessParameter.HeatBalances.v_t]);
      REAL2REAL_107 : REAL2REAL;
      REAL2REAL_112 : REAL2REAL;
      to_HeatBalances1 : PUBLISH_6(QI := 1, ID := 127.0.0.1:64501);
      from_ESCADA27 : SUBSCRIBE_1(QI := 1, ID := sfp[ProcessParameter.HeatBalances.h]);
      REAL2REAL_109 : REAL2REAL;
      REAL2REAL_111 : REAL2REAL;
      REAL2REAL_113 : REAL2REAL;
      from_ESCADA30 : SUBSCRIBE_1(QI := 1, ID := sfp[ProcessParameter.HeatBalances.theta_out]);
      REAL2REAL_116 : REAL2REAL;
      REAL2REAL_117 : REAL2REAL;
      from_ESCADA33 : SUBSCRIBE_1(QI := 1, ID := sfp[ProcessParameter.HeatBalances.Cp1]);
      REAL2REAL_118 : REAL2REAL;
      from_ESCADA32 : SUBSCRIBE_1(QI := 1, ID := sfp[ProcessParameter.HeatBalances.Cp_w1]);
      from_ESCADA31 : SUBSCRIBE_1(QI := 1, ID := sfp[ProcessParameter.HeatBalances.Cp_c]);
      REAL2REAL_114 : REAL2REAL;
      from_ESCADA29 : SUBSCRIBE_1(QI := 1, ID := sfp[ProcessParameter.HeatBalances.K_loss]);
      from_ESCADA34 : SUBSCRIBE_1(QI := 1, ID := sfp[ProcessParameter.HeatBalances.K_loss1]);
      to_HeatBalances2 : PUBLISH_6(QI := 1, ID := 127.0.0.1:64502);
      REAL2REAL_115 : REAL2REAL;
      REAL2REAL_120 : REAL2REAL;
      from_ESCADA35 : SUBSCRIBE_1(QI := 1, ID := sfp[ProcessParameter.HeatBalances.Cp_met]);
      to_HeatBalances3 : PUBLISH_4(QI := 1, ID := 127.0.0.1:64503);
      from_ESCADA36 : SUBSCRIBE_1(QI := 1, ID := sfp[ProcessParameter.HeatBalances.theta_acc]);
      REAL2REAL_122 : REAL2REAL;
      REAL2REAL_121 : REAL2REAL;
      from_ESCADA37 : SUBSCRIBE_1(QI := 1, ID := sfp[ProcessParameter.HeatBalances.Cp_c1]);
      from_ESCADA38 : SUBSCRIBE_1(QI := 1, ID := sfp[ProcessParameter.HeatBalances.Cp_w2]);
      REAL2REAL_119 : REAL2REAL;
      REAL2REAL_123 : REAL2REAL;
      from_ESCADA41 : SUBSCRIBE_1(QI := 1, ID := sfp[ProcessParameter.DifferentialPressureBalances.K_ce]);
      REAL2REAL_125 : REAL2REAL;
      REAL2REAL_124 : REAL2REAL;
      to_DifferentialPressureBalances : PUBLISH_3(QI := 1, ID := 127.0.0.1:64600);
      from_ESCADA40 : SUBSCRIBE_1(QI := 1, ID := sfp[ProcessParameter.DifferentialPressureBalances.K_c]);
      from_ESCADA39 : SUBSCRIBE_1(QI := 1, ID := sfp[ProcessParameter.DifferentialPressureBalances.K_auf]);
      from_ESCADA45 : SUBSCRIBE_1(QI := 1, ID := sfp[ProcessParameter.PowerBalances.M_on]);
      from_ESCADA42 : SUBSCRIBE_1(QI := 1, ID := sfp[ProcessParameter.PowerBalances.K_power]);
      from_ESCADA43 : SUBSCRIBE_1(QI := 1, ID := sfp[ProcessParameter.PowerBalances.w]);
      REAL2REAL_128_0 : REAL2REAL;
      to_PowerBalances1 : PUBLISH_4(QI := 1, ID := 127.0.0.1:64701);
      from_ESCADA44 : SUBSCRIBE_1(QI := 1, ID := sfp[ProcessParameter.PowerBalances.N_rol]);
      REAL2REAL_126 : REAL2REAL;
      REAL2REAL_129_0 : REAL2REAL;
      REAL2REAL_127_0 : REAL2REAL;
      from_ESCADA47 : SUBSCRIBE_1(QI := 1, ID := sfp[ProcessParameter.PowerBalances.P_f]);
      REAL2REAL_131 : REAL2REAL;
      from_ESCADA46 : SUBSCRIBE_1(QI := 1, ID := sfp[ProcessParameter.PowerBalances.M_v]);
      REAL2REAL_132 : REAL2REAL;
      REAL2REAL_130 : REAL2REAL;
      to_PowerBalances2 : PUBLISH_3(QI := 1, ID := 127.0.0.1:64702);
      from_ESCADA48 : SUBSCRIBE_1(QI := 1, ID := sfp[ProcessParameter.PowerBalances.K_g]);
      SUBSCRIBE_1 : SUBSCRIBE_1(QI := 1, ID := sfp[START_BOOL]);
      BOOL2BOOL : BOOL2BOOL;
      PUBLISH_1 : PUBLISH_1(QI := 1, ID := 127.0.0.1:30000);
      PUBLISH_1_0 : PUBLISH_1(QI := 1, ID := 127.0.0.1:10000);
      PUBLISH_1_1 : PUBLISH_1(QI := 1, ID := 127.0.0.1:20000);
      PUBLISH_1_2 : PUBLISH_1(QI := 1, ID := 127.0.0.1:40000);
      PUBLISH_1_3 : PUBLISH_1(QI := 1, ID := 127.0.0.1:50000);
      PUBLISH_1_4 : PUBLISH_1(QI := 1, ID := 127.0.0.1:60000);
      PUBLISH_1_5 : PUBLISH_1(QI := 1, ID := 127.0.0.1:70000);
    END_FBS
    EVENT_CONNECTIONS
      from_GrindingZone.IND TO REAL2REAL_68.REQ;
      from_GrindingZone.IND TO REAL2REAL_69.REQ;
      REAL2REAL_68.CNF TO to_ESCADA2.REQ;
      REAL2REAL_69.CNF TO to_ESCADA3.REQ;
      from_GrindingZone.INITO TO to_ESCADA2.INIT;
      from_GrindingZone.INITO TO to_ESCADA3.INIT;
      START.COLD TO from_GrindingZone.INIT;
      START.WARM TO from_GrindingZone.INIT;
      from_SeparatorZone.IND TO REAL2REAL_74.REQ;
      from_SeparatorZone.IND TO REAL2REAL_72.REQ;
      REAL2REAL_73.CNF TO to_ESCADA7.REQ;
      REAL2REAL_71.CNF TO to_ESCADA5.REQ;
      from_SeparatorZone.IND TO REAL2REAL_73.REQ;
      from_SeparatorZone.IND TO REAL2REAL_71.REQ;
      from_SeparatorZone.IND TO REAL2REAL_70.REQ;
      REAL2REAL_72.CNF TO to_ESCADA6.REQ;
      REAL2REAL_70.CNF TO to_ESCADA4.REQ;
      REAL2REAL_74.CNF TO to_ESCADA8.REQ;
      from_SeparatorZone.INITO TO to_ESCADA4.INIT;
      from_SeparatorZone.INITO TO to_ESCADA5.INIT;
      from_SeparatorZone.INITO TO to_ESCADA6.INIT;
      from_SeparatorZone.INITO TO to_ESCADA7.INIT;
      from_SeparatorZone.INITO TO to_ESCADA8.INIT;
      START.COLD TO from_SeparatorZone.INIT;
      START.WARM TO from_SeparatorZone.INIT;
      REAL2REAL_76.CNF TO tp_ESCADA10.REQ;
      REAL2REAL_75.CNF TO to_ESCADA9.REQ;
      from_ClassifierZone.IND TO REAL2REAL_76.REQ;
      from_ClassifierZone.IND TO REAL2REAL_78.REQ;
      from_ClassifierZone.IND TO REAL2REAL_75.REQ;
      REAL2REAL_77.CNF TO to_ESCADA11.REQ;
      REAL2REAL_78.CNF TO to_ESCADA12.REQ;
      from_ClassifierZone.IND TO REAL2REAL_77.REQ;
      from_ClassifierZone.INITO TO to_ESCADA9.INIT;
      from_ClassifierZone.INITO TO tp_ESCADA10.INIT;
      from_ClassifierZone.INITO TO to_ESCADA11.INIT;
      from_ClassifierZone.INITO TO to_ESCADA12.INIT;
      START.COLD TO from_ClassifierZone.INIT;
      START.WARM TO from_ClassifierZone.INIT;
      REAL2REAL_79.CNF TO to_ESCADA13.REQ;
      from_HeatBalances.IND TO REAL2REAL_79.REQ;
      from_HeatBalances.INITO TO to_ESCADA13.INIT;
      START.COLD TO from_HeatBalances.INIT;
      START.WARM TO from_HeatBalances.INIT;
      from_DifferentialPressureBalances.IND TO REAL2REAL_80.REQ;
      REAL2REAL_80.CNF TO to_ESCADA14.REQ;
      from_DifferentialPressureBalances.INITO TO to_ESCADA14.INIT;
      START.COLD TO from_DifferentialPressureBalances.INIT;
      START.WARM TO from_DifferentialPressureBalances.INIT;
      from_PowerBalances.IND TO REAL2REAL_81.REQ;
      from_PowerBalances.IND TO REAL2REAL_83.REQ;
      REAL2REAL_82.CNF TO to_ESCADA16.REQ;
      from_PowerBalances.IND TO REAL2REAL_82.REQ;
      REAL2REAL_83.CNF TO to_ESCADA17.REQ;
      REAL2REAL_81.CNF TO to_ESCADA15.REQ;
      from_PowerBalances.INITO TO to_ESCADA15.INIT;
      from_PowerBalances.INITO TO to_ESCADA16.INIT;
      from_PowerBalances.INITO TO to_ESCADA17.INIT;
      START.COLD TO from_PowerBalances.INIT;
      START.WARM TO from_PowerBalances.INIT;
      from_ESCADA.IND TO m_F.REQ;
      m_F.CNF TO to_BowlZone.REQ;
      from_ESCADA.INITO TO to_BowlZone.INIT;
      START.COLD TO from_ESCADA.INIT;
      START.WARM TO from_ESCADA.INIT;
      from_ESCADA1.IND TO REAL2REAL_85.REQ;
      REAL2REAL_85.CNF TO to_SeparatorZone.REQ;
      START.COLD TO from_ESCADA1.INIT;
      START.WARM TO from_ESCADA1.INIT;
      from_ESCADA1.INITO TO to_SeparatorZone.INIT;
      REAL2REAL_86.CNF TO to_HeatBalances.REQ;
      from_ESCADA3.IND TO REAL2REAL_87.REQ;
      REAL2REAL_88.CNF TO to_HeatBalances.REQ;
      REAL2REAL_89.CNF TO to_HeatBalances.REQ;
      from_ESCADA5.IND TO REAL2REAL_89.REQ;
      from_ESCADA2.IND TO REAL2REAL_86.REQ;
      from_ESCADA4.IND TO REAL2REAL_88.REQ;
      REAL2REAL_87.CNF TO to_HeatBalances.REQ;
      from_ESCADA2.INITO TO to_HeatBalances.INIT;
      START.COLD TO from_ESCADA4.INIT;
      START.WARM TO from_ESCADA4.INIT;
      START.COLD TO from_ESCADA5.INIT;
      START.WARM TO from_ESCADA5.INIT;
      START.COLD TO from_ESCADA2.INIT;
      START.WARM TO from_ESCADA2.INIT;
      START.COLD TO from_ESCADA3.INIT;
      START.WARM TO from_ESCADA3.INIT;
      from_ESCADA6.IND TO REAL2REAL_90.REQ;
      REAL2REAL_90.CNF TO to_PowerBalances.REQ;
      from_ESCADA6.INITO TO to_PowerBalances.INIT;
      START.COLD TO from_ESCADA6.INIT;
      START.WARM TO from_ESCADA6.INIT;
      from_ESCADA7.IND TO a_i.REQ;
      from_ESCADA8.IND TO t_BG.REQ;
      a_i.CNF TO to_BowlZone2.REQ;
      t_BG.CNF TO to_BowlZone2.REQ;
      from_ESCADA8.INITO TO to_BowlZone2.INIT;
      START.COLD TO from_ESCADA8.INIT;
      START.WARM TO from_ESCADA8.INIT;
      START.COLD TO from_ESCADA7.INIT;
      START.WARM TO from_ESCADA7.INIT;
      from_ESCADA12.IND TO REAL2REAL_96.REQ;
      REAL2REAL_95.CNF TO to_GrindingZone.REQ;
      REAL2REAL_96.CNF TO to_GrindingZone.REQ;
      from_ESCADA11.IND TO REAL2REAL_95.REQ;
      REAL2REAL_93.CNF TO to_GrindingZone.REQ;
      from_ESCADA10.IND TO REAL2REAL_94.REQ;
      from_ESCADA9.IND TO REAL2REAL_93.REQ;
      REAL2REAL_94.CNF TO to_GrindingZone.REQ;
      from_ESCADA9.INITO TO to_GrindingZone.INIT;
      START.COLD TO from_ESCADA10.INIT;
      START.WARM TO from_ESCADA10.INIT;
      START.COLD TO from_ESCADA11.INIT;
      START.WARM TO from_ESCADA11.INIT;
      START.COLD TO from_ESCADA12.INIT;
      START.WARM TO from_ESCADA12.INIT;
      START.COLD TO from_ESCADA9.INIT;
      START.WARM TO from_ESCADA9.INIT;
      REAL2REAL_97.CNF TO to_SeparatorZone1.REQ;
      REAL2REAL_99.CNF TO to_SeparatorZone1.REQ;
      REAL2REAL_100.CNF TO to_SeparatorZone1.REQ;
      REAL2REAL_102.CNF TO to_SeparatorZone1.REQ;
      from_ESCADA15.IND TO REAL2REAL_99.REQ;
      from_ESCADA17.IND TO REAL2REAL_101.REQ;
      from_ESCADA14.IND TO REAL2REAL_98.REQ;
      from_ESCADA18.IND TO REAL2REAL_102.REQ;
      from_ESCADA16.IND TO REAL2REAL_100.REQ;
      REAL2REAL_98.CNF TO to_SeparatorZone1.REQ;
      REAL2REAL_101.CNF TO to_SeparatorZone1.REQ;
      from_ESCADA13.IND TO REAL2REAL_97.REQ;
      from_ESCADA13.INITO TO to_SeparatorZone1.INIT;
      START.COLD TO from_ESCADA16.INIT;
      START.WARM TO from_ESCADA16.INIT;
      START.COLD TO from_ESCADA15.INIT;
      START.WARM TO from_ESCADA15.INIT;
      START.COLD TO from_ESCADA14.INIT;
      START.WARM TO from_ESCADA14.INIT;
      START.COLD TO from_ESCADA17.INIT;
      START.WARM TO from_ESCADA17.INIT;
      START.COLD TO from_ESCADA18.INIT;
      START.WARM TO from_ESCADA18.INIT;
      START.COLD TO from_ESCADA13.INIT;
      START.WARM TO from_ESCADA13.INIT;
      REAL2REAL_103.CNF TO to_ClassifierZone.REQ;
      REAL2REAL_105.CNF TO to_ClassifierZone.REQ;
      from_ESCADA19.IND TO REAL2REAL_103.REQ;
      REAL2REAL_104.CNF TO to_ClassifierZone.REQ;
      from_ESCADA22.IND TO REAL2REAL_106.REQ;
      REAL2REAL_106.CNF TO to_ClassifierZone.REQ;
      from_ESCADA21.IND TO REAL2REAL_105.REQ;
      from_ESCADA20.IND TO REAL2REAL_104.REQ;
      from_ESCADA19.INITO TO to_ClassifierZone.INIT;
      START.COLD TO from_ESCADA22.INIT;
      START.WARM TO from_ESCADA22.INIT;
      START.COLD TO from_ESCADA20.INIT;
      START.WARM TO from_ESCADA20.INIT;
      START.COLD TO from_ESCADA19.INIT;
      START.WARM TO from_ESCADA19.INIT;
      START.COLD TO from_ESCADA21.INIT;
      START.WARM TO from_ESCADA21.INIT;
      REAL2REAL_112.CNF TO to_HeatBalances1.REQ;
      from_ESCADA24.IND TO REAL2REAL_108.REQ;
      from_ESCADA25.IND TO REAL2REAL_109.REQ;
      REAL2REAL_109.CNF TO to_HeatBalances1.REQ;
      REAL2REAL_108.CNF TO to_HeatBalances1.REQ;
      REAL2REAL_107.CNF TO to_HeatBalances1.REQ;
      from_ESCADA26.IND TO REAL2REAL_110.REQ;
      from_ESCADA28.IND TO REAL2REAL_112.REQ;
      from_ESCADA27.IND TO REAL2REAL_111.REQ;
      REAL2REAL_111.CNF TO to_HeatBalances1.REQ;
      from_ESCADA23.IND TO REAL2REAL_107.REQ;
      REAL2REAL_110.CNF TO to_HeatBalances1.REQ;
      from_ESCADA23.INITO TO to_HeatBalances1.INIT;
      START.COLD TO from_ESCADA26.INIT;
      START.WARM TO from_ESCADA26.INIT;
      START.COLD TO from_ESCADA24.INIT;
      START.WARM TO from_ESCADA24.INIT;
      START.COLD TO from_ESCADA23.INIT;
      START.WARM TO from_ESCADA23.INIT;
      START.COLD TO from_ESCADA25.INIT;
      START.WARM TO from_ESCADA25.INIT;
      START.COLD TO from_ESCADA28.INIT;
      START.WARM TO from_ESCADA28.INIT;
      START.COLD TO from_ESCADA27.INIT;
      START.WARM TO from_ESCADA27.INIT;
      REAL2REAL_115.CNF TO to_HeatBalances2.REQ;
      from_ESCADA31.IND TO REAL2REAL_115.REQ;
      from_ESCADA34.IND TO REAL2REAL_118.REQ;
      from_ESCADA32.IND TO REAL2REAL_116.REQ;
      from_ESCADA33.IND TO REAL2REAL_117.REQ;
      from_ESCADA30.IND TO REAL2REAL_114.REQ;
      REAL2REAL_114.CNF TO to_HeatBalances2.REQ;
      REAL2REAL_118.CNF TO to_HeatBalances2.REQ;
      REAL2REAL_117.CNF TO to_HeatBalances2.REQ;
      from_ESCADA29.IND TO REAL2REAL_113.REQ;
      REAL2REAL_116.CNF TO to_HeatBalances2.REQ;
      REAL2REAL_113.CNF TO to_HeatBalances2.REQ;
      from_ESCADA29.INITO TO to_HeatBalances2.INIT;
      START.COLD TO from_ESCADA30.INIT;
      START.WARM TO from_ESCADA30.INIT;
      START.COLD TO from_ESCADA33.INIT;
      START.WARM TO from_ESCADA33.INIT;
      START.COLD TO from_ESCADA32.INIT;
      START.WARM TO from_ESCADA32.INIT;
      START.COLD TO from_ESCADA31.INIT;
      START.WARM TO from_ESCADA31.INIT;
      START.COLD TO from_ESCADA29.INIT;
      START.WARM TO from_ESCADA29.INIT;
      START.COLD TO from_ESCADA34.INIT;
      START.WARM TO from_ESCADA34.INIT;
      REAL2REAL_122.CNF TO to_HeatBalances3.REQ;
      REAL2REAL_119.CNF TO to_HeatBalances3.REQ;
      REAL2REAL_120.CNF TO to_HeatBalances3.REQ;
      from_ESCADA36.IND TO REAL2REAL_120.REQ;
      REAL2REAL_121.CNF TO to_HeatBalances3.REQ;
      from_ESCADA38.IND TO REAL2REAL_122.REQ;
      from_ESCADA35.IND TO REAL2REAL_119.REQ;
      from_ESCADA37.IND TO REAL2REAL_121.REQ;
      from_ESCADA35.INITO TO to_HeatBalances3.INIT;
      START.COLD TO from_ESCADA35.INIT;
      START.WARM TO from_ESCADA35.INIT;
      START.COLD TO from_ESCADA36.INIT;
      START.WARM TO from_ESCADA36.INIT;
      START.COLD TO from_ESCADA37.INIT;
      START.WARM TO from_ESCADA37.INIT;
      START.COLD TO from_ESCADA38.INIT;
      START.WARM TO from_ESCADA38.INIT;
      from_ESCADA41.IND TO REAL2REAL_125.REQ;
      from_ESCADA40.IND TO REAL2REAL_124.REQ;
      REAL2REAL_123.CNF TO to_DifferentialPressureBalances.REQ;
      REAL2REAL_124.CNF TO to_DifferentialPressureBalances.REQ;
      REAL2REAL_125.CNF TO to_DifferentialPressureBalances.REQ;
      from_ESCADA39.IND TO REAL2REAL_123.REQ;
      from_ESCADA39.INITO TO to_DifferentialPressureBalances.INIT;
      START.COLD TO from_ESCADA41.INIT;
      START.WARM TO from_ESCADA41.INIT;
      START.COLD TO from_ESCADA40.INIT;
      START.WARM TO from_ESCADA40.INIT;
      START.COLD TO from_ESCADA39.INIT;
      START.WARM TO from_ESCADA39.INIT;
      REAL2REAL_129_0.CNF TO to_PowerBalances1.REQ;
      REAL2REAL_127_0.CNF TO to_PowerBalances1.REQ;
      from_ESCADA43.IND TO REAL2REAL_127_0.REQ;
      from_ESCADA42.IND TO REAL2REAL_126.REQ;
      from_ESCADA44.IND TO REAL2REAL_128_0.REQ;
      from_ESCADA45.IND TO REAL2REAL_129_0.REQ;
      REAL2REAL_126.CNF TO to_PowerBalances1.REQ;
      REAL2REAL_128_0.CNF TO to_PowerBalances1.REQ;
      from_ESCADA42.INITO TO to_PowerBalances1.INIT;
      START.COLD TO from_ESCADA45.INIT;
      START.WARM TO from_ESCADA45.INIT;
      START.COLD TO from_ESCADA42.INIT;
      START.WARM TO from_ESCADA42.INIT;
      START.COLD TO from_ESCADA43.INIT;
      START.WARM TO from_ESCADA43.INIT;
      START.COLD TO from_ESCADA44.INIT;
      START.WARM TO from_ESCADA44.INIT;
      REAL2REAL_131.CNF TO to_PowerBalances2.REQ;
      from_ESCADA48.IND TO REAL2REAL_132.REQ;
      REAL2REAL_132.CNF TO to_PowerBalances2.REQ;
      REAL2REAL_130.CNF TO to_PowerBalances2.REQ;
      from_ESCADA46.IND TO REAL2REAL_130.REQ;
      from_ESCADA47.IND TO REAL2REAL_131.REQ;
      from_ESCADA46.INITO TO to_PowerBalances2.INIT;
      START.COLD TO from_ESCADA47.INIT;
      START.WARM TO from_ESCADA47.INIT;
      START.COLD TO from_ESCADA46.INIT;
      START.WARM TO from_ESCADA46.INIT;
      START.COLD TO from_ESCADA48.INIT;
      START.WARM TO from_ESCADA48.INIT;
      SUBSCRIBE_1.IND TO BOOL2BOOL.REQ;
      START.COLD TO SUBSCRIBE_1.INIT;
      START.WARM TO SUBSCRIBE_1.INIT;
      BOOL2BOOL.CNF TO PUBLISH_1_0.REQ;
      BOOL2BOOL.CNF TO PUBLISH_1_1.REQ;
      BOOL2BOOL.CNF TO PUBLISH_1.REQ;
      SUBSCRIBE_1.INITO TO PUBLISH_1_0.INIT;
      SUBSCRIBE_1.INITO TO PUBLISH_1_1.INIT;
      SUBSCRIBE_1.INITO TO PUBLISH_1.INIT;
      BOOL2BOOL.CNF TO PUBLISH_1_2.REQ;
      SUBSCRIBE_1.INITO TO PUBLISH_1_2.INIT;
      BOOL2BOOL.CNF TO PUBLISH_1_3.REQ;
      SUBSCRIBE_1.INITO TO PUBLISH_1_3.INIT;
      BOOL2BOOL.CNF TO PUBLISH_1_4.REQ;
      SUBSCRIBE_1.INITO TO PUBLISH_1_4.INIT;
      BOOL2BOOL.CNF TO PUBLISH_1_5.REQ;
      SUBSCRIBE_1.INITO TO PUBLISH_1_5.INIT;
    END_CONNECTIONS
    DATA_CONNECTIONS
      from_GrindingZone.RD_2 TO REAL2REAL_69.IN;
      REAL2REAL_68.OUT TO to_ESCADA2.SD_1;
      REAL2REAL_69.OUT TO to_ESCADA3.SD_1;
      from_GrindingZone.RD_1 TO REAL2REAL_68.IN;
      REAL2REAL_74.OUT TO to_ESCADA8.SD_1;
      REAL2REAL_72.OUT TO to_ESCADA6.SD_1;
      REAL2REAL_70.OUT TO to_ESCADA4.SD_1;
      from_SeparatorZone.RD_1 TO REAL2REAL_70.IN;
      from_SeparatorZone.RD_4 TO REAL2REAL_73.IN;
      from_SeparatorZone.RD_2 TO REAL2REAL_71.IN;
      from_SeparatorZone.RD_5 TO REAL2REAL_74.IN;
      REAL2REAL_73.OUT TO to_ESCADA7.SD_1;
      from_SeparatorZone.RD_3 TO REAL2REAL_72.IN;
      REAL2REAL_71.OUT TO to_ESCADA5.SD_1;
      REAL2REAL_76.OUT TO tp_ESCADA10.SD_1;
      REAL2REAL_77.OUT TO to_ESCADA11.SD_1;
      from_ClassifierZone.RD_2 TO REAL2REAL_76.IN;
      from_ClassifierZone.RD_1 TO REAL2REAL_75.IN;
      from_ClassifierZone.RD_4 TO REAL2REAL_78.IN;
      REAL2REAL_75.OUT TO to_ESCADA9.SD_1;
      from_ClassifierZone.RD_3 TO REAL2REAL_77.IN;
      REAL2REAL_78.OUT TO to_ESCADA12.SD_1;
      from_HeatBalances.RD_1 TO REAL2REAL_79.IN;
      REAL2REAL_79.OUT TO to_ESCADA13.SD_1;
      REAL2REAL_80.OUT TO to_ESCADA14.SD_1;
      from_DifferentialPressureBalances.RD_1 TO REAL2REAL_80.IN;
      REAL2REAL_81.OUT TO to_ESCADA15.SD_1;
      from_PowerBalances.RD_2 TO REAL2REAL_82.IN;
      from_PowerBalances.RD_3 TO REAL2REAL_83.IN;
      REAL2REAL_83.OUT TO to_ESCADA17.SD_1;
      REAL2REAL_82.OUT TO to_ESCADA16.SD_1;
      from_PowerBalances.RD_1 TO REAL2REAL_81.IN;
      from_ESCADA.RD_1 TO m_F.IN;
      m_F.OUT TO to_BowlZone.SD_1;
      REAL2REAL_85.OUT TO to_SeparatorZone.SD_1;
      from_ESCADA1.RD_1 TO REAL2REAL_85.IN;
      REAL2REAL_87.OUT TO to_HeatBalances.SD_2;
      from_ESCADA2.RD_1 TO REAL2REAL_86.IN;
      from_ESCADA4.RD_1 TO REAL2REAL_88.IN;
      REAL2REAL_89.OUT TO to_HeatBalances.SD_4;
      from_ESCADA3.RD_1 TO REAL2REAL_87.IN;
      REAL2REAL_86.OUT TO to_HeatBalances.SD_1;
      REAL2REAL_88.OUT TO to_HeatBalances.SD_3;
      from_ESCADA5.RD_1 TO REAL2REAL_89.IN;
      REAL2REAL_90.OUT TO to_PowerBalances.SD_1;
      from_ESCADA6.RD_1 TO REAL2REAL_90.IN;
      from_ESCADA7.RD_1 TO a_i.IN;
      a_i.OUT TO to_BowlZone2.SD_1;
      from_ESCADA8.RD_1 TO t_BG.IN;
      t_BG.OUT TO to_BowlZone2.SD_2;
      REAL2REAL_96.OUT TO to_GrindingZone.SD_4;
      REAL2REAL_94.OUT TO to_GrindingZone.SD_2;
      from_ESCADA10.RD_1 TO REAL2REAL_94.IN;
      REAL2REAL_95.OUT TO to_GrindingZone.SD_3;
      REAL2REAL_93.OUT TO to_GrindingZone.SD_1;
      from_ESCADA12.RD_1 TO REAL2REAL_96.IN;
      from_ESCADA11.RD_1 TO REAL2REAL_95.IN;
      from_ESCADA9.RD_1 TO REAL2REAL_93.IN;
      REAL2REAL_98.OUT TO to_SeparatorZone1.SD_2;
      from_ESCADA16.RD_1 TO REAL2REAL_100.IN;
      REAL2REAL_100.OUT TO to_SeparatorZone1.SD_4;
      REAL2REAL_102.OUT TO to_SeparatorZone1.SD_6;
      from_ESCADA17.RD_1 TO REAL2REAL_101.IN;
      from_ESCADA15.RD_1 TO REAL2REAL_99.IN;
      REAL2REAL_99.OUT TO to_SeparatorZone1.SD_3;
      REAL2REAL_97.OUT TO to_SeparatorZone1.SD_1;
      from_ESCADA14.RD_1 TO REAL2REAL_98.IN;
      from_ESCADA13.RD_1 TO REAL2REAL_97.IN;
      REAL2REAL_101.OUT TO to_SeparatorZone1.SD_5;
      from_ESCADA18.RD_1 TO REAL2REAL_102.IN;
      REAL2REAL_104.OUT TO to_ClassifierZone.SD_2;
      from_ESCADA19.RD_1 TO REAL2REAL_103.IN;
      REAL2REAL_103.OUT TO to_ClassifierZone.SD_1;
      from_ESCADA20.RD_1 TO REAL2REAL_104.IN;
      from_ESCADA22.RD_1 TO REAL2REAL_106.IN;
      REAL2REAL_105.OUT TO to_ClassifierZone.SD_3;
      from_ESCADA21.RD_1 TO REAL2REAL_105.IN;
      REAL2REAL_106.OUT TO to_ClassifierZone.SD_4;
      from_ESCADA25.RD_1 TO REAL2REAL_109.IN;
      REAL2REAL_108.OUT TO to_HeatBalances1.SD_2;
      REAL2REAL_110.OUT TO to_HeatBalances1.SD_4;
      from_ESCADA28.RD_1 TO REAL2REAL_112.IN;
      from_ESCADA26.RD_1 TO REAL2REAL_110.IN;
      from_ESCADA24.RD_1 TO REAL2REAL_108.IN;
      REAL2REAL_112.OUT TO to_HeatBalances1.SD_6;
      REAL2REAL_107.OUT TO to_HeatBalances1.SD_1;
      REAL2REAL_111.OUT TO to_HeatBalances1.SD_5;
      REAL2REAL_109.OUT TO to_HeatBalances1.SD_3;
      from_ESCADA27.RD_1 TO REAL2REAL_111.IN;
      from_ESCADA23.RD_1 TO REAL2REAL_107.IN;
      REAL2REAL_113.OUT TO to_HeatBalances2.SD_1;
      from_ESCADA34.RD_1 TO REAL2REAL_118.IN;
      REAL2REAL_117.OUT TO to_HeatBalances2.SD_5;
      from_ESCADA31.RD_1 TO REAL2REAL_115.IN;
      from_ESCADA33.RD_1 TO REAL2REAL_117.IN;
      REAL2REAL_116.OUT TO to_HeatBalances2.SD_4;
      REAL2REAL_114.OUT TO to_HeatBalances2.SD_2;
      REAL2REAL_118.OUT TO to_HeatBalances2.SD_6;
      from_ESCADA29.RD_1 TO REAL2REAL_113.IN;
      from_ESCADA30.RD_1 TO REAL2REAL_114.IN;
      from_ESCADA32.RD_1 TO REAL2REAL_116.IN;
      REAL2REAL_115.OUT TO to_HeatBalances2.SD_3;
      from_ESCADA36.RD_1 TO REAL2REAL_120.IN;
      REAL2REAL_121.OUT TO to_HeatBalances3.SD_3;
      from_ESCADA37.RD_1 TO REAL2REAL_121.IN;
      from_ESCADA35.RD_1 TO REAL2REAL_119.IN;
      REAL2REAL_122.OUT TO to_HeatBalances3.SD_4;
      REAL2REAL_119.OUT TO to_HeatBalances3.SD_1;
      REAL2REAL_120.OUT TO to_HeatBalances3.SD_2;
      from_ESCADA38.RD_1 TO REAL2REAL_122.IN;
      REAL2REAL_125.OUT TO to_DifferentialPressureBalances.SD_3;
      REAL2REAL_124.OUT TO to_DifferentialPressureBalances.SD_2;
      from_ESCADA41.RD_1 TO REAL2REAL_125.IN;
      from_ESCADA39.RD_1 TO REAL2REAL_123.IN;
      from_ESCADA40.RD_1 TO REAL2REAL_124.IN;
      REAL2REAL_123.OUT TO to_DifferentialPressureBalances.SD_1;
      from_ESCADA45.RD_1 TO REAL2REAL_129_0.IN;
      REAL2REAL_129_0.OUT TO to_PowerBalances1.SD_4;
      REAL2REAL_127_0.OUT TO to_PowerBalances1.SD_2;
      from_ESCADA42.RD_1 TO REAL2REAL_126.IN;
      from_ESCADA44.RD_1 TO REAL2REAL_128_0.IN;
      REAL2REAL_128_0.OUT TO to_PowerBalances1.SD_3;
      REAL2REAL_126.OUT TO to_PowerBalances1.SD_1;
      from_ESCADA43.RD_1 TO REAL2REAL_127_0.IN;
      from_ESCADA46.RD_1 TO REAL2REAL_130.IN;
      REAL2REAL_132.OUT TO to_PowerBalances2.SD_3;
      REAL2REAL_130.OUT TO to_PowerBalances2.SD_1;
      REAL2REAL_131.OUT TO to_PowerBalances2.SD_2;
      from_ESCADA47.RD_1 TO REAL2REAL_131.IN;
      from_ESCADA48.RD_1 TO REAL2REAL_132.IN;
      SUBSCRIBE_1.RD_1 TO BOOL2BOOL.IN;
      BOOL2BOOL.OUT TO PUBLISH_1_0.SD_1;
      BOOL2BOOL.OUT TO PUBLISH_1_1.SD_1;
      BOOL2BOOL.OUT TO PUBLISH_1.SD_1;
      BOOL2BOOL.OUT TO PUBLISH_1_2.SD_1;
      BOOL2BOOL.OUT TO PUBLISH_1_3.SD_1;
      BOOL2BOOL.OUT TO PUBLISH_1_4.SD_1;
      BOOL2BOOL.OUT TO PUBLISH_1_5.SD_1;
    END_CONNECTIONS
  END_APPLICATION
  DEVICE Process_Simulator : FORTE_PC(MGR_ID := "localhost:61499")
    {SET_ATTRIBUTE(Profile, HOLOBLOC)}
    RESOURCE EMB_RES : EMB_RES
      FBS
        mF : REAL2REAL(IN := 1);
        F_MUL : F_MUL;
        F_ADD : F_ADD;
        F_ADD_0 : F_ADD;
        F_SUB : F_SUB;
        REAL2REAL_0 : REAL2REAL;
        REAL2REAL_0_0 : REAL2REAL;
        REAL2REAL_0_1 : REAL2REAL;
        a1 : REAL2REAL(IN := 0.5);
        m_SB : REAL2REAL(IN := 1);
        m_CB : REAL2REAL(IN := 1);
        E_CYCLE : E_CYCLE(DT := T#200ms);
        FB_INTEGRATE : FB_INTEGRATE(K := 1);
        REAL2REAL_0_1_0 : REAL2REAL;
        M_B2 : REAL2REAL;
        F_DIV : F_DIV;
        mBG : REAL2REAL;
        tauBG : REAL2REAL(IN := 0.5);
        MV_from_ESCADA : SUBSCRIBE_1(QI := 1, ID := 127.0.0.1:63100);
        PP_from_ESCADA1 : SUBSCRIBE_2(QI := 1, ID := 127.0.0.1:64100);
        START_Subscribe : SUBSCRIBE_1(QI := 1, ID := 127.0.0.1:10000);
        E_SWITCH_0 : E_SWITCH;
        m_BG : REAL2REAL(IN := 1);
        gamma1 : REAL2REAL(IN := 0.5);
        bJ : REAL2REAL(IN := 0.5);
        gammaJ : REAL2REAL(IN := 0.5);
        F_ADD_1 : F_ADD;
        REAL2REAL_2_0 : REAL2REAL;
        F_SUB_0 : F_SUB;
        FB_INTEGRATE_0 : FB_INTEGRATE(K := 1);
        REAL2REAL_2_0_0 : REAL2REAL;
        F_DIV_0 : F_DIV;
        tauGS : REAL2REAL(IN := 0.5);
        mGS : REAL2REAL;
        E_CYCLE_0 : E_CYCLE(DT := T#200ms);
        F_MUL_1 : F_MUL;
        F_MUL_1_2 : F_MUL;
        F_MUL_1_3 : F_MUL;
        REAL2REAL_2_0_3 : REAL2REAL;
        F_SUB_0_0 : F_SUB;
        REAL2REAL_2_0_3_0 : REAL2REAL;
        REAL2REAL_2_0_3_1 : REAL2REAL;
        REAL2REAL_2_0_3_0_0 : REAL2REAL;
        M_G2 : REAL2REAL;
        to_InputOutput1 : PUBLISH_2(QI := 1, ID := 127.0.0.1:62200);
        from_EclipseScada5 : SUBSCRIBE_4(QI := 1, ID := 127.0.0.1:64200);
        SUBSCRIBE_1_2 : SUBSCRIBE_1(QI := 1, ID := 127.0.0.1:20000);
        E_SWITCH_1 : E_SWITCH;
        m_air_inC : REAL2REAL(IN := 1);
        Cons1_0 : REAL2REAL(IN := 0.5959);
        F_MUL_2_1 : F_MUL;
        F_MUL_2_0_1 : F_MUL;
        REAL2REAL_2_1 : REAL2REAL;
        F_MUL_2_0_0_0 : F_MUL;
        Cons2_0 : REAL2REAL(IN := 22.69);
        REAL2REAL_2_2_1 : REAL2REAL;
        REAL2REAL_2_2_0_0 : REAL2REAL;
        F_SUB_1_0 : F_SUB;
        Cons3_0 : REAL2REAL(IN := 311.36);
        F_ADD_2_0 : F_ADD;
        REAL2REAL_2_2_0_1_0 : REAL2REAL;
        c2 : REAL2REAL;
        REAL2REAL_2_2_1_0_1 : REAL2REAL;
        F_SUB_2_1 : F_SUB;
        F_MUL_5_0 : F_MUL;
        cons4_0 : REAL2REAL(IN := 0.001);
        REAL2REAL_2_2_1_0_0_0 : REAL2REAL;
        d_min_0 : REAL2REAL(IN := 0.25);
        F_SUB_2_0_0 : F_SUB;
        d_max_0 : REAL2REAL(IN := 0.5);
        REAL2REAL_2_2_1_1_0 : REAL2REAL;
        REAL2REAL_2_2_1_2_0 : REAL2REAL;
        F_DIV_4 : F_DIV;
        m_SC : REAL2REAL(IN := 1);
        tau_CFU : REAL2REAL(IN := 0.5);
        tau_CB : REAL2REAL(IN := 0.5);
        m_AirIN : REAL2REAL(IN := 1);
        F_ADD_3_0 : F_ADD;
        REAL2REAL_21 : REAL2REAL;
        F_SUB_4_0 : F_SUB;
        REAL2REAL_8_0 : REAL2REAL;
        F_SUB_4_0_0 : F_SUB;
        REAL2REAL_8_0_0 : REAL2REAL;
        FB_INTEGRATE_2 : FB_INTEGRATE(K := 1);
        F_MUL_7 : F_MUL;
        REAL2REAL_10_0 : REAL2REAL;
        F_DIV_5 : F_DIV;
        mCFU : REAL2REAL;
        F_SUB_7_0 : F_SUB;
        REAL2REAL_10_0_0 : REAL2REAL(IN := 1);
        F_MUL_7_0 : F_MUL;
        REAL2REAL_10_1 : REAL2REAL;
        F_DIV_5_0 : F_DIV;
        mCB : REAL2REAL;
        REAL2REAL_10_0_0_0 : REAL2REAL;
        E_CYCLE_2 : E_CYCLE(DT := T#200ms);
        M_C2 : REAL2REAL;
        m_air_outC : REAL2REAL;
        to_InputOutput3 : PUBLISH_4(QI := 1, ID := 127.0.0.1:62400);
        SUBSCRIBE_1_3 : SUBSCRIBE_1(QI := 1, ID := 127.0.0.1:40000);
        E_SWITCH_2 : E_SWITCH;
        from_EclipseScada7 : SUBSCRIBE_4(QI := 1, ID := 127.0.0.1:64400);
        E_CYCLE_3 : E_CYCLE(DT := T#200ms);
        m_airS : REAL2REAL(IN := 1);
        Cp_a : REAL2REAL(IN := 0.5);
        T_m_air : REAL2REAL(IN := 25);
        F_MUL_0 : F_MUL;
        REAL2REAL_1_0 : REAL2REAL;
        F_MUL_8 : F_MUL;
        REAL2REAL_4_0 : REAL2REAL;
        m_CF : REAL2REAL(IN := 1);
        Satu : REAL2REAL(IN := 1);
        theta_FB : REAL2REAL(IN := 0.5);
        Cp : REAL2REAL(IN := 0.5);
        T_a : REAL2REAL(IN := 25);
        F_SUB_6 : F_SUB;
        F_MUL_9 : F_MUL;
        REAL2REAL_6_0 : REAL2REAL;
        F_MUL_10 : F_MUL;
        REAL2REAL_9_0 : REAL2REAL;
        REAL2REAL_11_0 : REAL2REAL;
        F_MUL_11 : F_MUL;
        REAL2REAL_12_0 : REAL2REAL;
        Cp_w : REAL2REAL(IN := 0.5);
        F_MUL_12 : F_MUL;
        F_MUL_13 : F_MUL;
        REAL2REAL_13_0 : REAL2REAL;
        REAL2REAL_14_0 : REAL2REAL;
        F_MUL_14 : F_MUL;
        REAL2REAL_15_0 : REAL2REAL;
        Hg : REAL2REAL(IN := 5);
        m_mois : REAL2REAL(IN := 1);
        h : REAL2REAL(IN := 0.5);
        v_t : REAL2REAL(IN := 0.5);
        F_MUL_13_0 : F_MUL;
        REAL2REAL_16_0 : REAL2REAL;
        F_MUL_17 : F_MUL;
        REAL2REAL_17_0 : REAL2REAL;
        K_loss : REAL2REAL(IN := 0.5);
        F_MUL_15_0 : F_MUL;
        REAL2REAL_18_0 : REAL2REAL;
        F_ADD_4 : F_ADD;
        REAL2REAL_19_0 : REAL2REAL;
        F_ADD_5 : F_ADD;
        REAL2REAL_20_0 : REAL2REAL;
        F_SUB_8 : F_SUB;
        REAL2REAL_21_0 : REAL2REAL;
        F_ADD_6 : F_ADD;
        REAL2REAL_22_0 : REAL2REAL;
        F_ADD_7 : F_ADD;
        REAL2REAL_23_0 : REAL2REAL;
        m_CFU : REAL2REAL(IN := 1);
        Satu1 : REAL2REAL(IN := 1);
        theta_out : REAL2REAL(IN := 0.5);
        Cp_c : REAL2REAL(IN := 0.5);
        F_SUB_9 : F_SUB;
        REAL2REAL_24_0 : REAL2REAL;
        F_MUL_16_0 : F_MUL;
        REAL2REAL_25_0 : REAL2REAL;
        F_MUL_18_0 : F_MUL;
        REAL2REAL_26_0 : REAL2REAL;
        F_MUL_19_0 : F_MUL;
        REAL2REAL_27_0 : REAL2REAL;
        Cp_w1 : REAL2REAL(IN := 0.5);
        F_MUL_20_0 : F_MUL;
        REAL2REAL_29_0 : REAL2REAL;
        F_MUL_21_0 : F_MUL;
        REAL2REAL_30_0 : REAL2REAL;
        F_MUL_22_0 : F_MUL;
        REAL2REAL_31_0 : REAL2REAL;
        Cp1 : REAL2REAL(IN := 0.5);
        F_MUL_24_0 : F_MUL;
        REAL2REAL_28_0 : REAL2REAL;
        F_MUL_25_0 : F_MUL;
        REAL2REAL_32_0 : REAL2REAL;
        K_loss1 : REAL2REAL(IN := 1);
        F_MUL_23_0 : F_MUL;
        REAL2REAL_33_0 : REAL2REAL;
        REAL2REAL_34_0 : REAL2REAL;
        F_ADD_8 : F_ADD;
        REAL2REAL_35_0 : REAL2REAL;
        F_ADD_9 : F_ADD;
        REAL2REAL_36_0 : REAL2REAL;
        F_SUB_11 : F_SUB;
        REAL2REAL_37_0 : REAL2REAL;
        M_met : REAL2REAL(IN := 1);
        Cp_met : REAL2REAL(IN := 0.5);
        F_MUL_26_0 : F_MUL;
        REAL2REAL_38_0 : REAL2REAL;
        M_B : REAL2REAL(IN := 1);
        M_G : REAL2REAL(IN := 1);
        M_C : REAL2REAL(IN := 1);
        F_ADD_10 : F_ADD;
        REAL2REAL_39_0 : REAL2REAL;
        F_ADD_11 : F_ADD;
        REAL2REAL_40_0 : REAL2REAL;
        REAL2REAL_41_0 : REAL2REAL;
        Satu2 : REAL2REAL(IN := 1);
        theta_acc : REAL2REAL(IN := 0.5);
        F_SUB_12 : F_SUB;
        Cp_c1 : REAL2REAL(IN := 0.5);
        F_MUL_27_0 : F_MUL;
        REAL2REAL_42_0 : REAL2REAL;
        F_MUL_28_0 : F_MUL;
        REAL2REAL_43_0 : REAL2REAL;
        F_ADD_12 : F_ADD;
        REAL2REAL_44_0 : REAL2REAL;
        F_ADD_13 : F_ADD;
        REAL2REAL_45_0 : REAL2REAL;
        F_MUL_29_0 : F_MUL;
        REAL2REAL_46_0 : REAL2REAL;
        Cp_w2 : REAL2REAL(IN := 0.5);
        F_MUL_30_0 : F_MUL;
        REAL2REAL_47_0 : REAL2REAL;
        F_ADD_14 : F_ADD;
        REAL2REAL_48_0 : REAL2REAL;
        F_ADD_15 : F_ADD;
        REAL2REAL_49_0 : REAL2REAL;
        F_DIV_6 : F_DIV;
        dT_out : REAL2REAL;
        FB_INTEGRATE_3 : FB_INTEGRATE(K := 1);
        T_out : REAL2REAL;
        to_InputOutput4 : PUBLISH_1(QI := 1, ID := 127.0.0.1:62500);
        from_EclipseScada2 : SUBSCRIBE_4(QI := 1, ID := 127.0.0.1:63500);
        SUBSCRIBE_1_4 : SUBSCRIBE_1(QI := 1, ID := 127.0.0.1:50000);
        E_SWITCH_3 : E_SWITCH;
        from_EclipseScada8 : SUBSCRIBE_6(QI := 1, ID := 127.0.0.1:64501);
        from_EclipseScada9 : SUBSCRIBE_6(QI := 1, ID := 127.0.0.1:64502);
        from_EclipseScada10 : SUBSCRIBE_4(QI := 1, ID := 127.0.0.1:64503);
        F_ADD_3 : F_ADD;
        E_CYCLE_4 : E_CYCLE(DT := T#200ms);
        K_auf : REAL2REAL(IN := 0.5);
        m_airS1 : REAL2REAL(IN := 1);
        F_MUL_31 : F_MUL;
        REAL2REAL_52 : REAL2REAL;
        F_MUL_32 : F_MUL;
        REAL2REAL_53 : REAL2REAL;
        K_c : REAL2REAL(IN := 0.5);
        M_B1 : REAL2REAL(IN := 1);
        M_G1 : REAL2REAL(IN := 1);
        F_ADD_16 : F_ADD;
        REAL2REAL_54 : REAL2REAL;
        m_airS2 : REAL2REAL(IN := 1);
        F_MUL_33 : F_MUL;
        REAL2REAL_55 : REAL2REAL;
        F_MUL_34 : F_MUL;
        REAL2REAL_56 : REAL2REAL;
        F_MUL_35 : F_MUL;
        REAL2REAL_57 : REAL2REAL;
        K_ce : REAL2REAL(IN := 0.5);
        M_S : REAL2REAL(IN := 1);
        M_C1 : REAL2REAL(IN := 1);
        m_airS3 : REAL2REAL(IN := 1);
        F_MUL_36 : F_MUL;
        REAL2REAL_58 : REAL2REAL;
        F_ADD_17 : F_ADD;
        REAL2REAL_59 : REAL2REAL;
        F_MUL_37 : F_MUL;
        REAL2REAL_60 : REAL2REAL;
        F_MUL_38 : F_MUL;
        REAL2REAL_61 : REAL2REAL;
        F_ADD_18 : F_ADD;
        REAL2REAL_62 : REAL2REAL;
        F_ADD_19 : F_ADD;
        dP_mill : REAL2REAL;
        to_InputOutput5 : PUBLISH_1(QI := 1, ID := 127.0.0.1:62600);
        SUBSCRIBE_1_5 : SUBSCRIBE_1(QI := 1, ID := 127.0.0.1:60000);
        E_SWITCH_4 : E_SWITCH;
        from_EclipseScada11 : SUBSCRIBE_3(QI := 1, ID := 127.0.0.1:64600);
        K_power : REAL2REAL(IN := 0.5);
        M_G3 : REAL2REAL(IN := 2);
        w : REAL2REAL(IN := 1);
        N_rol : REAL2REAL(IN := 0.5);
        F_MUL_39 : F_MUL;
        REAL2REAL_50 : REAL2REAL;
        F_MUL_40 : F_MUL;
        REAL2REAL_51 : REAL2REAL;
        F_MUL_41 : F_MUL;
        REAL2REAL_63 : REAL2REAL;
        P_load : REAL2REAL(IN := 2);
        F_ADD_20 : F_ADD;
        REAL2REAL_64 : REAL2REAL;
        M_on : REAL2REAL(IN := 1);
        F_MUL_42 : F_MUL;
        P_total : REAL2REAL;
        M_v : REAL2REAL(IN := 0.5);
        P_f : REAL2REAL(IN := 0.5);
        F_MUL_43 : F_MUL;
        REAL2REAL_66 : REAL2REAL;
        F_DIV_7 : F_DIV;
        I_total : REAL2REAL;
        K_g : REAL2REAL(IN := 0.5);
        F_MUL_44 : F_MUL;
        Hg1 : REAL2REAL;
        E_CYCLE_5 : E_CYCLE(DT := T#200ms);
        to_InputOutput6 : PUBLISH_3(QI := 1, ID := 127.0.0.1:62700);
        from_EclipseScada3 : SUBSCRIBE_1(QI := 1, ID := 127.0.0.1:63700);
        SUBSCRIBE_1_6 : SUBSCRIBE_1(QI := 1, ID := 127.0.0.1:70000);
        E_SWITCH_5 : E_SWITCH;
        from_EclipseScada12 : SUBSCRIBE_4(QI := 1, ID := 127.0.0.1:64701);
        from_EclipseScada13 : SUBSCRIBE_3(QI := 1, ID := 127.0.0.1:64702);
        m_air_inS_plus_noise : REAL2REAL;
        Cons1 : REAL2REAL(IN := 0.5728);
        F_MUL_2 : F_MUL;
        F_MUL_2_0 : F_MUL;
        REAL2REAL_2 : REAL2REAL;
        F_MUL_2_0_0 : F_MUL;
        Cons2 : REAL2REAL(IN := 14.307);
        REAL2REAL_2_2 : REAL2REAL;
        REAL2REAL_2_2_0 : REAL2REAL;
        F_SUB_1 : F_SUB;
        Cons3 : REAL2REAL(IN := 180.22);
        F_ADD_2 : F_ADD;
        REAL2REAL_2_2_0_1 : REAL2REAL;
        c1 : REAL2REAL;
        REAL2REAL_2_2_1_0 : REAL2REAL;
        F_SUB_2 : F_SUB;
        F_MUL_5 : F_MUL;
        cons4 : REAL2REAL(IN := 0.001);
        REAL2REAL_2_2_1_0_0 : REAL2REAL;
        d_min : REAL2REAL(IN := 0.25);
        F_SUB_2_0 : F_SUB;
        d_max : REAL2REAL(IN := 0.5);
        REAL2REAL_2_2_1_1 : REAL2REAL;
        REAL2REAL_2_2_1_2 : REAL2REAL;
        m_GS : REAL2REAL(IN := 1);
        rho : REAL2REAL(IN := 0.5);
        nu_acc : REAL2REAL(IN := 0.5);
        F_MUL_3_0 : F_MUL;
        F_MUL_4_0 : F_MUL;
        REAL2REAL_5_0 : REAL2REAL;
        m_mois1 : REAL2REAL;
        F_SUB_3_0 : F_SUB;
        REAL2REAL_5_0_0 : REAL2REAL;
        F_SUB_3_0_0 : F_SUB;
        REAL2REAL_5_0_0_0 : REAL2REAL;
        F_SUB_3_0_0_0 : F_SUB;
        REAL2REAL_5_0_0_0_0 : REAL2REAL;
        FB_INTEGRATE_1 : FB_INTEGRATE(K := 1);
        F_MUL_6_0 : F_MUL;
        REAL2REAL_7_0 : REAL2REAL;
        tauSC : REAL2REAL(IN := 0.5);
        tauSB : REAL2REAL(IN := 0.5);
        REAL2REAL_3_0 : REAL2REAL(IN := 1);
        F_SUB_5_0 : F_SUB;
        F_MUL_6_0_0 : F_MUL;
        REAL2REAL_7_0_0 : REAL2REAL;
        REAL2REAL_7_1 : REAL2REAL;
        F_DIV_1 : F_DIV;
        F_DIV_2 : F_DIV;
        mSC : REAL2REAL;
        mSB : REAL2REAL;
        E_CYCLE_1 : E_CYCLE(DT := T#200ms);
        F_DIV_3 : F_DIV;
        M_S1 : REAL2REAL;
        m_air_outS : REAL2REAL;
        m_air_inS : REAL2REAL(IN := 1);
        to_InputOutput2 : PUBLISH_5(QI := 1, ID := 127.0.0.1:62300);
        from_EclipseScada1 : SUBSCRIBE_1(QI := 1, ID := 127.0.0.1:63300);
        from_EclipseScada6 : SUBSCRIBE_6(QI := 1, ID := 127.0.0.1:64300);
        SUBSCRIBE_1_0 : SUBSCRIBE_1(QI := 1, ID := 127.0.0.1:30000);
        E_SWITCH : E_SWITCH;
      END_FBS
      EVENT_CONNECTIONS
        START.COLD TO FB_INTEGRATE.INIT;
        START.WARM TO FB_INTEGRATE.INIT;
        START.COLD TO FB_INTEGRATE_0.INIT;
        START.WARM TO FB_INTEGRATE_0.INIT;
        START.COLD TO FB_INTEGRATE_2.INIT;
        START.WARM TO FB_INTEGRATE_2.INIT;
        START.COLD TO FB_INTEGRATE_3.INIT;
        START.WARM TO FB_INTEGRATE_3.INIT;
        START.COLD TO FB_INTEGRATE_1.INIT;
        START.WARM TO FB_INTEGRATE_1.INIT;
        START.COLD TO to_InputOutput5.INIT;
        START.WARM TO to_InputOutput5.INIT;
        START.COLD TO to_InputOutput6.INIT;
        START.WARM TO to_InputOutput6.INIT;
        START.COLD TO MV_from_ESCADA.INIT;
        START.WARM TO MV_from_ESCADA.INIT;
        START.COLD TO from_EclipseScada1.INIT;
        START.WARM TO from_EclipseScada1.INIT;
        START.COLD TO from_EclipseScada2.INIT;
        START.WARM TO from_EclipseScada2.INIT;
        START.COLD TO from_EclipseScada3.INIT;
        START.WARM TO from_EclipseScada3.INIT;
        START.COLD TO PP_from_ESCADA1.INIT;
        START.WARM TO PP_from_ESCADA1.INIT;
        START.COLD TO from_EclipseScada5.INIT;
        START.WARM TO from_EclipseScada5.INIT;
        START.COLD TO from_EclipseScada6.INIT;
        START.WARM TO from_EclipseScada6.INIT;
        START.COLD TO SUBSCRIBE_1_0.INIT;
        START.WARM TO SUBSCRIBE_1_0.INIT;
        START.COLD TO START_Subscribe.INIT;
        START.WARM TO START_Subscribe.INIT;
        START.COLD TO SUBSCRIBE_1_2.INIT;
        START.WARM TO SUBSCRIBE_1_2.INIT;
        START.COLD TO SUBSCRIBE_1_3.INIT;
        START.WARM TO SUBSCRIBE_1_3.INIT;
        START.COLD TO from_EclipseScada7.INIT;
        START.WARM TO from_EclipseScada7.INIT;
        START.COLD TO SUBSCRIBE_1_4.INIT;
        START.WARM TO SUBSCRIBE_1_4.INIT;
        START.COLD TO from_EclipseScada8.INIT;
        START.WARM TO from_EclipseScada8.INIT;
        START.COLD TO from_EclipseScada9.INIT;
        START.WARM TO from_EclipseScada9.INIT;
        START.COLD TO from_EclipseScada10.INIT;
        START.WARM TO from_EclipseScada10.INIT;
        START.COLD TO SUBSCRIBE_1_5.INIT;
        START.WARM TO SUBSCRIBE_1_5.INIT;
        START.COLD TO from_EclipseScada11.INIT;
        START.WARM TO from_EclipseScada11.INIT;
        START.COLD TO SUBSCRIBE_1_6.INIT;
        START.WARM TO SUBSCRIBE_1_6.INIT;
        START.COLD TO from_EclipseScada12.INIT;
        START.WARM TO from_EclipseScada12.INIT;
        START.COLD TO from_EclipseScada13.INIT;
        START.WARM TO from_EclipseScada13.INIT;
        M_B2.CNF TO F_DIV.REQ;
        FB_INTEGRATE.CNF TO M_B2.REQ;
        F_SUB.CNF TO REAL2REAL_0_1_0.REQ;
        F_MUL.CNF TO REAL2REAL_0.REQ;
        REAL2REAL_0_1_0.CNF TO FB_INTEGRATE.REQ;
        F_ADD_0.CNF TO REAL2REAL_0_1.REQ;
        F_ADD.CNF TO REAL2REAL_0_0.REQ;
        REAL2REAL_0.CNF TO F_ADD.REQ;
        E_CYCLE.EO TO m_SB.REQ;
        REAL2REAL_0_0.CNF TO F_ADD_0.REQ;
        REAL2REAL_0_1.CNF TO F_SUB.REQ;
        E_CYCLE.EO TO tauBG.REQ;
        E_CYCLE.EO TO mF.REQ;
        E_CYCLE.EO TO m_CB.REQ;
        F_DIV.CNF TO mBG.REQ;
        E_CYCLE.EO TO a1.REQ;
        mF.CNF TO F_MUL.REQ;
        START_Subscribe.IND TO E_SWITCH_0.EI;
        E_SWITCH_0.EO1 TO E_CYCLE.START;
        REAL2REAL_2_0.CNF TO F_SUB_0.REQ;
        m_BG.CNF TO F_ADD_1.REQ;
        E_CYCLE_0.EO TO tauGS.REQ;
        F_MUL_1_3.CNF TO REAL2REAL_2_0_3_1.REQ;
        F_SUB_0_0.CNF TO REAL2REAL_2_0_3_0_0.REQ;
        E_CYCLE_0.EO TO bJ.REQ;
        F_ADD_1.CNF TO REAL2REAL_2_0.REQ;
        REAL2REAL_2_0_3.CNF TO F_MUL_1_3.REQ;
        REAL2REAL_2_0_0.CNF TO FB_INTEGRATE_0.REQ;
        F_DIV_0.CNF TO mGS.REQ;
        REAL2REAL_2_0_3_0.CNF TO F_SUB_0_0.REQ;
        F_MUL_1_2.CNF TO REAL2REAL_2_0_3.REQ;
        FB_INTEGRATE_0.CNF TO F_MUL_1_2.REQ;
        FB_INTEGRATE_0.CNF TO F_DIV_0.REQ;
        E_CYCLE_0.EO TO m_BG.REQ;
        FB_INTEGRATE_0.CNF TO M_G2.REQ;
        FB_INTEGRATE_0.CNF TO F_MUL_1.REQ;
        F_MUL_1.CNF TO REAL2REAL_2_0_3_0.REQ;
        F_SUB_0.CNF TO REAL2REAL_2_0_0.REQ;
        E_CYCLE_0.EO TO gammaJ.REQ;
        E_CYCLE_0.EO TO gamma1.REQ;
        mGS.CNF TO to_InputOutput1.REQ;
        FB_INTEGRATE_0.INITO TO to_InputOutput1.INIT;
        SUBSCRIBE_1_2.IND TO E_SWITCH_1.EI;
        E_SWITCH_1.EO1 TO E_CYCLE_0.START;
        REAL2REAL_2_2_0_1_0.CNF TO F_ADD_2_0.REQ;
        FB_INTEGRATE_2.CNF TO M_C2.REQ;
        E_CYCLE_2.EO TO m_SC.REQ;
        REAL2REAL_10_0.CNF TO F_DIV_5.REQ;
        E_CYCLE_2.EO TO tau_CFU.REQ;
        F_MUL_2_0_1.CNF TO REAL2REAL_2_1.REQ;
        REAL2REAL_21.CNF TO F_SUB_4_0.REQ;
        REAL2REAL_10_0_0_0.CNF TO F_MUL_7_0.REQ;
        REAL2REAL_2_2_1_0_0_0.CNF TO F_SUB_2_1.REQ;
        REAL2REAL_8_0_0.CNF TO FB_INTEGRATE_2.REQ;
        Cons2_0.CNF TO F_MUL_2_0_0_0.REQ;
        F_SUB_2_0_0.CNF TO REAL2REAL_2_2_1_1_0.REQ;
        F_SUB_2_1.CNF TO REAL2REAL_2_2_1_2_0.REQ;
        F_DIV_5_0.CNF TO mCB.REQ;
        E_CYCLE_2.EO TO Cons1_0.REQ;
        F_ADD_2_0.CNF TO cons4_0.REQ;
        FB_INTEGRATE_2.CNF TO REAL2REAL_10_0_0_0.REQ;
        m_air_inC.CNF TO m_air_outC.REQ;
        F_MUL_2_1.CNF TO REAL2REAL_2_2_0_0.REQ;
        c2.CNF TO REAL2REAL_10_0_0.REQ;
        F_DIV_5.CNF TO mCFU.REQ;
        F_SUB_1_0.CNF TO REAL2REAL_2_2_0_1_0.REQ;
        F_SUB_4_0.CNF TO REAL2REAL_8_0.REQ;
        E_CYCLE_2.EO TO m_air_inC.REQ;
        c2.CNF TO F_SUB_7_0.REQ;
        F_MUL_5_0.CNF TO d_min_0.REQ;
        REAL2REAL_8_0.CNF TO F_SUB_4_0_0.REQ;
        FB_INTEGRATE_2.CNF TO F_MUL_7.REQ;
        E_CYCLE_2.EO TO Cons2_0.REQ;
        F_DIV_4.CNF TO c2.REQ;
        m_air_inC.CNF TO F_MUL_2_0_1.REQ;
        F_ADD_3_0.CNF TO REAL2REAL_21.REQ;
        F_MUL_7_0.CNF TO REAL2REAL_10_1.REQ;
        F_MUL_2_0_0_0.CNF TO REAL2REAL_2_2_1.REQ;
        REAL2REAL_2_2_1_0_0_0.CNF TO F_SUB_2_0_0.REQ;
        F_SUB_4_0_0.CNF TO REAL2REAL_8_0_0.REQ;
        REAL2REAL_2_1.CNF TO F_MUL_2_1.REQ;
        E_CYCLE_2.EO TO m_AirIN.REQ;
        F_MUL_7.CNF TO REAL2REAL_10_0.REQ;
        REAL2REAL_2_2_1_0_1.CNF TO F_MUL_5_0.REQ;
        m_AirIN.CNF TO F_ADD_3_0.REQ;
        REAL2REAL_2_2_1_2_0.CNF TO F_DIV_4.REQ;
        REAL2REAL_10_1.CNF TO F_DIV_5_0.REQ;
        F_ADD_2_0.CNF TO REAL2REAL_2_2_1_0_1.REQ;
        E_CYCLE_2.EO TO Cons3_0.REQ;
        F_MUL_5_0.CNF TO d_max_0.REQ;
        E_CYCLE_2.EO TO tau_CB.REQ;
        REAL2REAL_2_2_0_0.CNF TO F_SUB_1_0.REQ;
        F_MUL_5_0.CNF TO REAL2REAL_2_2_1_0_0_0.REQ;
        mCFU.CNF TO to_InputOutput3.REQ;
        FB_INTEGRATE_2.INITO TO to_InputOutput3.INIT;
        SUBSCRIBE_1_3.IND TO E_SWITCH_2.EI;
        E_SWITCH_2.EO1 TO E_CYCLE_2.START;
        F_MUL_21_0.CNF TO REAL2REAL_30_0.REQ;
        dT_out.CNF TO FB_INTEGRATE_3.REQ;
        F_MUL_30_0.CNF TO REAL2REAL_47_0.REQ;
        Cp_w.CNF TO F_MUL_13.REQ;
        F_MUL_11.CNF TO REAL2REAL_12_0.REQ;
        F_MUL_28_0.CNF TO REAL2REAL_43_0.REQ;
        F_SUB_6.CNF TO REAL2REAL_6_0.REQ;
        F_MUL_20_0.CNF TO REAL2REAL_29_0.REQ;
        F_ADD_13.CNF TO REAL2REAL_45_0.REQ;
        E_CYCLE_3.EO TO M_B.REQ;
        Cp_c.CNF TO F_MUL_18_0.REQ;
        REAL2REAL_37_0.CNF TO F_DIV_6.REQ;
        K_loss.CNF TO F_MUL_15_0.REQ;
        REAL2REAL_42_0.CNF TO F_MUL_28_0.REQ;
        F_MUL_16_0.CNF TO REAL2REAL_25_0.REQ;
        REAL2REAL_40_0.CNF TO F_MUL_27_0.REQ;
        Satu.CNF TO F_SUB_6.REQ;
        E_CYCLE_3.EO TO Cp_c.REQ;
        M_met.CNF TO F_MUL_26_0.REQ;
        F_ADD_15.CNF TO REAL2REAL_49_0.REQ;
        M_B.CNF TO F_ADD_10.REQ;
        F_MUL_12.CNF TO REAL2REAL_13_0.REQ;
        F_MUL_17.CNF TO REAL2REAL_17_0.REQ;
        E_CYCLE_3.EO TO theta_acc.REQ;
        F_MUL_22_0.CNF TO REAL2REAL_31_0.REQ;
        E_CYCLE_3.EO TO h.REQ;
        E_CYCLE_3.EO TO M_C.REQ;
        F_ADD_4.CNF TO REAL2REAL_19_0.REQ;
        E_CYCLE_3.EO TO Satu.REQ;
        REAL2REAL_22_0.CNF TO F_ADD_7.REQ;
        E_CYCLE_3.EO TO T_a.REQ;
        m_mois.CNF TO F_MUL_13_0.REQ;
        m_airS.CNF TO F_MUL_0.REQ;
        E_CYCLE_3.EO TO M_met.REQ;
        m_CF.CNF TO F_MUL_12.REQ;
        F_MUL_29_0.CNF TO REAL2REAL_46_0.REQ;
        F_MUL_18_0.CNF TO REAL2REAL_26_0.REQ;
        F_ADD_12.CNF TO REAL2REAL_44_0.REQ;
        F_SUB_9.CNF TO REAL2REAL_24_0.REQ;
        E_CYCLE_3.EO TO Cp1.REQ;
        F_MUL_23_0.CNF TO REAL2REAL_33_0.REQ;
        REAL2REAL_44_0.CNF TO F_ADD_13.REQ;
        REAL2REAL_29_0.CNF TO F_MUL_22_0.REQ;
        REAL2REAL_25_0.CNF TO F_MUL_19_0.REQ;
        E_CYCLE_3.EO TO Cp.REQ;
        E_CYCLE_3.EO TO m_CFU.REQ;
        E_CYCLE_3.EO TO Cp_met.REQ;
        REAL2REAL_16_0.CNF TO F_MUL_17.REQ;
        REAL2REAL_46_0.CNF TO F_MUL_30_0.REQ;
        REAL2REAL_48_0.CNF TO F_ADD_15.REQ;
        E_CYCLE_3.EO TO m_CF.REQ;
        F_MUL_14.CNF TO REAL2REAL_15_0.REQ;
        F_MUL_9.CNF TO REAL2REAL_9_0.REQ;
        F_MUL_8.CNF TO REAL2REAL_4_0.REQ;
        E_CYCLE_3.EO TO m_mois.REQ;
        E_CYCLE_3.EO TO theta_out.REQ;
        REAL2REAL_17_0.CNF TO F_SUB_8.REQ;
        F_ADD_7.CNF TO REAL2REAL_23_0.REQ;
        Cp1.CNF TO F_MUL_24_0.REQ;
        F_SUB_8.CNF TO REAL2REAL_21_0.REQ;
        REAL2REAL_1_0.CNF TO F_MUL_8.REQ;
        E_CYCLE_3.EO TO Cp_c1.REQ;
        E_CYCLE_3.EO TO T_m_air.REQ;
        F_MUL_19_0.CNF TO REAL2REAL_27_0.REQ;
        REAL2REAL_15_0.CNF TO F_ADD_5.REQ;
        E_CYCLE_3.EO TO m_airS.REQ;
        F_MUL_24_0.CNF TO REAL2REAL_28_0.REQ;
        REAL2REAL_28_0.CNF TO F_MUL_25_0.REQ;
        F_MUL_13.CNF TO REAL2REAL_14_0.REQ;
        Satu2.CNF TO F_SUB_12.REQ;
        F_MUL_15_0.CNF TO REAL2REAL_18_0.REQ;
        REAL2REAL_9_0.CNF TO F_MUL_11.REQ;
        E_CYCLE_3.EO TO theta_FB.REQ;
        E_CYCLE_3.EO TO Cp_a.REQ;
        M_B.CNF TO F_ADD_12.REQ;
        E_CYCLE_3.EO TO M_G.REQ;
        E_CYCLE_3.EO TO Satu2.REQ;
        REAL2REAL_34_0.CNF TO F_ADD_9.REQ;
        E_CYCLE_3.EO TO K_loss.REQ;
        REAL2REAL_13_0.CNF TO F_MUL_14.REQ;
        REAL2REAL_6_0.CNF TO F_MUL_9.REQ;
        REAL2REAL_24_0.CNF TO F_MUL_16_0.REQ;
        F_MUL_0.CNF TO REAL2REAL_1_0.REQ;
        F_ADD_8.CNF TO REAL2REAL_35_0.REQ;
        E_CYCLE_3.EO TO Cp_w1.REQ;
        REAL2REAL_20_0.CNF TO F_ADD_6.REQ;
        E_CYCLE_3.EO TO K_loss1.REQ;
        F_MUL_25_0.CNF TO REAL2REAL_32_0.REQ;
        m_CFU.CNF TO F_MUL_20_0.REQ;
        REAL2REAL_39_0.CNF TO F_ADD_11.REQ;
        F_MUL_13_0.CNF TO REAL2REAL_16_0.REQ;
        F_ADD_11.CNF TO REAL2REAL_40_0.REQ;
        F_DIV_6.CNF TO dT_out.REQ;
        REAL2REAL_32_0.CNF TO F_ADD_8.REQ;
        FB_INTEGRATE_3.CNF TO T_out.REQ;
        K_loss1.CNF TO F_MUL_23_0.REQ;
        F_MUL_10.CNF TO REAL2REAL_11_0.REQ;
        F_MUL_27_0.CNF TO REAL2REAL_42_0.REQ;
        F_ADD_10.CNF TO REAL2REAL_39_0.REQ;
        F_ADD_14.CNF TO REAL2REAL_48_0.REQ;
        Cp_w1.CNF TO F_MUL_21_0.REQ;
        F_ADD_6.CNF TO REAL2REAL_22_0.REQ;
        F_SUB_11.CNF TO REAL2REAL_37_0.REQ;
        F_ADD_9.CNF TO REAL2REAL_36_0.REQ;
        E_CYCLE_3.EO TO Cp_w.REQ;
        REAL2REAL_4_0.CNF TO F_ADD_4.REQ;
        Cp.CNF TO F_MUL_10.REQ;
        Satu1.CNF TO F_SUB_9.REQ;
        REAL2REAL_45_0.CNF TO F_MUL_29_0.REQ;
        F_SUB_12.CNF TO REAL2REAL_41_0.REQ;
        REAL2REAL_43_0.CNF TO F_ADD_14.REQ;
        E_CYCLE_3.EO TO Satu1.REQ;
        REAL2REAL_23_0.CNF TO F_SUB_11.REQ;
        E_CYCLE_3.EO TO Cp_w2.REQ;
        F_ADD_5.CNF TO REAL2REAL_20_0.REQ;
        F_MUL_26_0.CNF TO REAL2REAL_38_0.REQ;
        E_CYCLE_3.EO TO v_t.REQ;
        E_CYCLE_3.EO TO Hg.REQ;
        T_out.CNF TO to_InputOutput4.REQ;
        FB_INTEGRATE_3.INITO TO to_InputOutput4.INIT;
        SUBSCRIBE_1_4.IND TO E_SWITCH_3.EI;
        E_SWITCH_3.EO1 TO E_CYCLE_3.START;
        REAL2REAL_27_0.CNF TO F_ADD_3.REQ;
        F_ADD_3.CNF TO REAL2REAL_34_0.REQ;
        REAL2REAL_62.CNF TO F_ADD_19.REQ;
        E_CYCLE_4.EO TO m_airS2.REQ;
        F_ADD_17.CNF TO REAL2REAL_59.REQ;
        F_MUL_36.CNF TO REAL2REAL_58.REQ;
